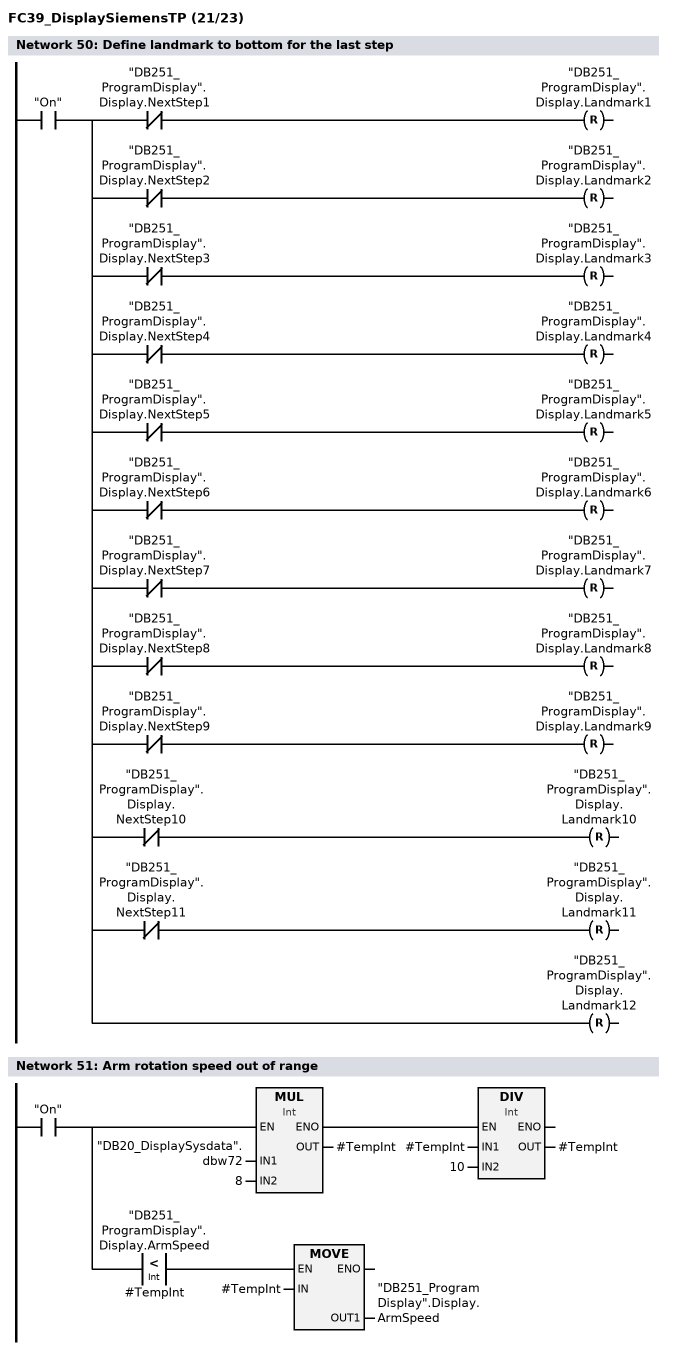
   RUNG wire#powerrail
      Contact( "On" )
      wire#w1
      I_Contact( "DB251_ProgramDisplay".Display.NextStep1 )
      R_Coil( "DB251_ProgramDisplay".Display.Landmark1 )
   END_RUNG
   RUNG wire#w1
      I_Contact( "DB251_ProgramDisplay".Display.NextStep2 )
      R_Coil( "DB251_ProgramDisplay".Display.Landmark2 )
   END_RUNG
   RUNG wire#w1
      I_Contact( "DB251_ProgramDisplay".Display.NextStep3 )
      R_Coil( "DB251_ProgramDisplay".Display.Landmark3 )
   END_RUNG
   RUNG wire#w1
      I_Contact( "DB251_ProgramDisplay".Display.NextStep4 )
      R_Coil( "DB251_ProgramDisplay".Display.Landmark4 )
   END_RUNG
   RUNG wire#w1
      I_Contact( "DB251_ProgramDisplay".Display.NextStep5 )
      R_Coil( "DB251_ProgramDisplay".Display.Landmark5 )
   END_RUNG
   RUNG wire#w1
      I_Contact( "DB251_ProgramDisplay".Display.NextStep6 )
      R_Coil( "DB251_ProgramDisplay".Display.Landmark6 )
   END_RUNG
   RUNG wire#w1
      I_Contact( "DB251_ProgramDisplay".Display.NextStep7 )
      R_Coil( "DB251_ProgramDisplay".Display.Landmark7 )
   END_RUNG
   RUNG wire#w1
      I_Contact( "DB251_ProgramDisplay".Display.NextStep8 )
      R_Coil( "DB251_ProgramDisplay".Display.Landmark8 )
   END_RUNG
   RUNG wire#w1
      I_Contact( "DB251_ProgramDisplay".Display.NextStep9 )
      R_Coil( "DB251_ProgramDisplay".Display.Landmark9 )
   END_RUNG
   RUNG wire#w1
      I_Contact( "DB251_ProgramDisplay".Display.NextStep10 )
      R_Coil( "DB251_ProgramDisplay".Display.Landmark10 )
   END_RUNG
   RUNG wire#w1
      I_Contact( "DB251_ProgramDisplay".Display.NextStep11 )
      R_Coil( "DB251_ProgramDisplay".Display.Landmark11 )
   END_RUNG
   RUNG wire#w1
      R_Coil( "DB251_ProgramDisplay".Display.Landmark12 )
   END_RUNG
   // the same network as SCL:
   IF "On" AND NOT "DB251_ProgramDisplay".Display.NextStep1 THEN
       "DB251_ProgramDisplay".Display.Landmark1 := FALSE;
   END_IF;
   IF "On" AND NOT "DB251_ProgramDisplay".Display.NextStep2 THEN
       "DB251_ProgramDisplay".Display.Landmark2 := FALSE;
   END_IF;
   IF "On" AND NOT "DB251_ProgramDisplay".Display.NextStep3 THEN
       "DB251_ProgramDisplay".Display.Landmark3 := FALSE;
   END_IF;
   IF "On" AND NOT "DB251_ProgramDisplay".Display.NextStep4 THEN
       "DB251_ProgramDisplay".Display.Landmark4 := FALSE;
   END_IF;
   IF "On" AND NOT "DB251_ProgramDisplay".Display.NextStep5 THEN
       "DB251_ProgramDisplay".Display.Landmark5 := FALSE;
   END_IF;
   IF "On" AND NOT "DB251_ProgramDisplay".Display.NextStep6 THEN
       "DB251_ProgramDisplay".Display.Landmark6 := FALSE;
   END_IF;
   IF "On" AND NOT "DB251_ProgramDisplay".Display.NextStep7 THEN
       "DB251_ProgramDisplay".Display.Landmark7 := FALSE;
   END_IF;
   IF "On" AND NOT "DB251_ProgramDisplay".Display.NextStep8 THEN
       "DB251_ProgramDisplay".Display.Landmark8 := FALSE;
   END_IF;
   IF "On" AND NOT "DB251_ProgramDisplay".Display.NextStep9 THEN
       "DB251_ProgramDisplay".Display.Landmark9 := FALSE;
   END_IF;
   IF "On" AND NOT "DB251_ProgramDisplay".Display.NextStep10 THEN
       "DB251_ProgramDisplay".Display.Landmark10 := FALSE;
   END_IF;
   IF "On" AND NOT "DB251_ProgramDisplay".Display.NextStep11 THEN
       "DB251_ProgramDisplay".Display.Landmark11 := FALSE;
   END_IF;
   IF "On" THEN "DB251_ProgramDisplay".Display.Landmark12 := FALSE; END_IF;
END_REGION

REGION Network 51: Arm rotation speed out of range
   RUNG wire#powerrail
      Contact( "On" )
      wire#w1
      { S7_Templates := "SrcType := Int"; S7_GenerateENO := "TRUE" } Mul(in1 := "DB20_DisplaySysdata".dbw72, in2 := 8, out => #TempInt)
      { S7_Templates := "SrcType := Int"; S7_GenerateENO := "TRUE" } Div(in1 := #TempInt, in2 := 10, out => #TempInt)
   END_RUNG
   RUNG wire#w1
      { S7_Templates := "SrcType := Int" } LT_Contact(in1 := "DB251_ProgramDisplay".Display.ArmSpeed, in2 := #TempInt)
      { S7_GenerateENO := "TRUE" } Move(in := #TempInt, out1 => "DB251_ProgramDisplay".Display.ArmSpeed)
   END_RUNG
   // the same network as SCL:
   // ENO of a box is taken as its EN; it also drops when the box reports an error
   IF "On" THEN
       #TempInt := "DB20_DisplaySysdata".dbw72 * 8;
       #TempInt := #TempInt / 10;
   END_IF;
   IF "On" AND ("DB251_ProgramDisplay".Display.ArmSpeed < #TempInt) THEN
       "DB251_ProgramDisplay".Display.ArmSpeed := #TempInt;
   END_IF;
END_REGION

REGION Network 52: Next step for spool carriage height 12 (0=End 1=Next)
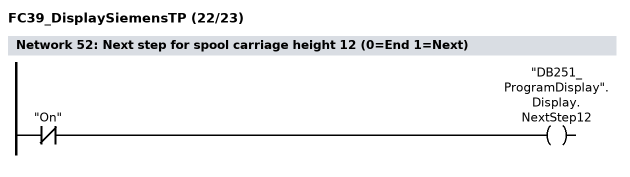
   RUNG wire#powerrail
      I_Contact( "On" )
      Coil( "DB251_ProgramDisplay".Display.NextStep12 )
   END_RUNG
   // the same network as SCL:
   "DB251_ProgramDisplay".Display.NextStep12 := NOT "On";
END_REGION

REGION Network 53
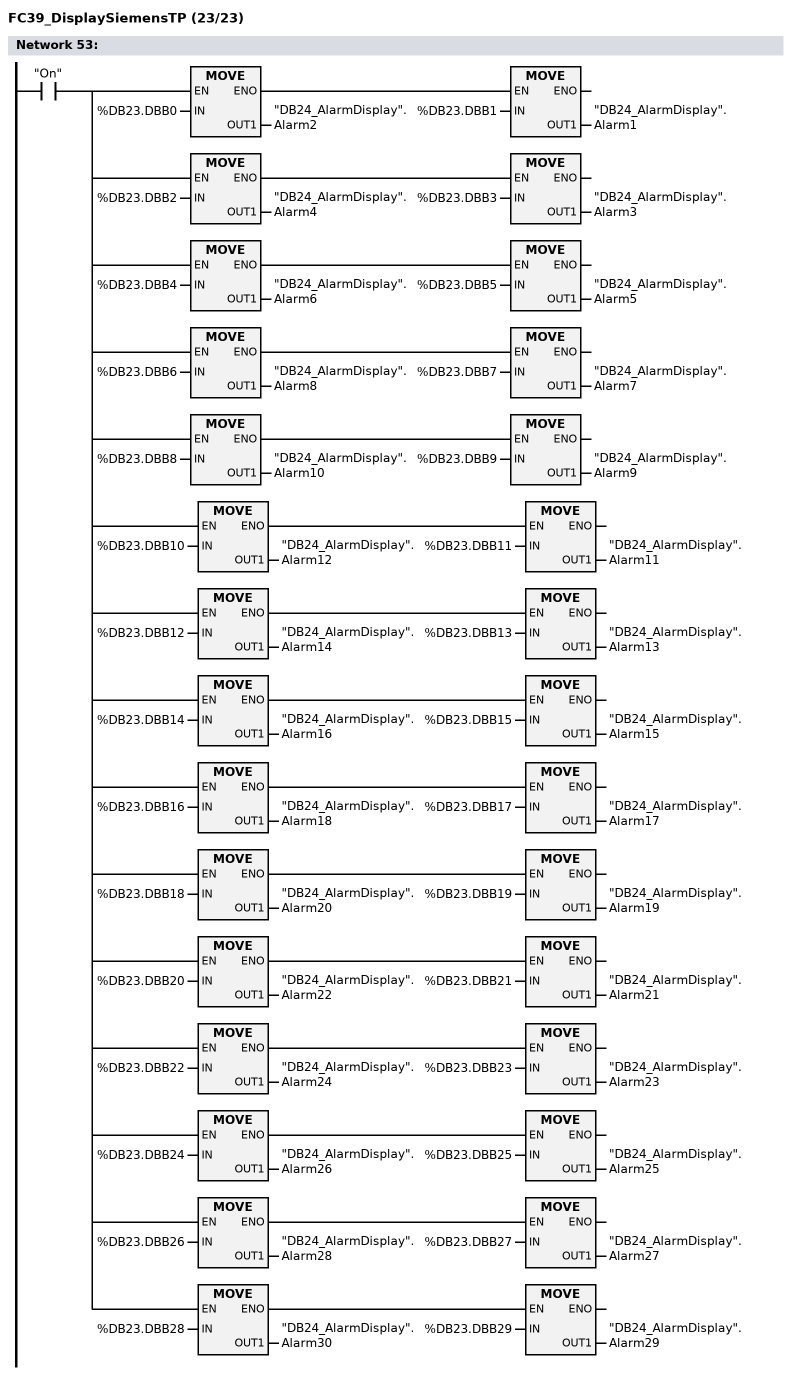
   RUNG wire#powerrail
      Contact( "On" )
      wire#w1
      { S7_GenerateENO := "TRUE" } Move(in := %DB23.DBB0, out1 => "DB24_AlarmDisplay".Alarm2)
      { S7_GenerateENO := "TRUE" } Move(in := %DB23.DBB1, out1 => "DB24_AlarmDisplay".Alarm1)
   END_RUNG
   RUNG wire#w1
      { S7_GenerateENO := "TRUE" } Move(in := %DB23.DBB2, out1 => "DB24_AlarmDisplay".Alarm4)
      { S7_GenerateENO := "TRUE" } Move(in := %DB23.DBB3, out1 => "DB24_AlarmDisplay".Alarm3)
   END_RUNG
   RUNG wire#w1
      { S7_GenerateENO := "TRUE" } Move(in := %DB23.DBB4, out1 => "DB24_AlarmDisplay".Alarm6)
      { S7_GenerateENO := "TRUE" } Move(in := %DB23.DBB5, out1 => "DB24_AlarmDisplay".Alarm5)
   END_RUNG
   RUNG wire#w1
      { S7_GenerateENO := "TRUE" } Move(in := %DB23.DBB6, out1 => "DB24_AlarmDisplay".Alarm8)
      { S7_GenerateENO := "TRUE" } Move(in := %DB23.DBB7, out1 => "DB24_AlarmDisplay".Alarm7)
   END_RUNG
   RUNG wire#w1
      { S7_GenerateENO := "TRUE" } Move(in := %DB23.DBB8, out1 => "DB24_AlarmDisplay".Alarm10)
      { S7_GenerateENO := "TRUE" } Move(in := %DB23.DBB9, out1 => "DB24_AlarmDisplay".Alarm9)
   END_RUNG
   RUNG wire#w1
      { S7_GenerateENO := "TRUE" } Move(in := %DB23.DBB10, out1 => "DB24_AlarmDisplay".Alarm12)
      { S7_GenerateENO := "TRUE" } Move(in := %DB23.DBB11, out1 => "DB24_AlarmDisplay".Alarm11)
   END_RUNG
   RUNG wire#w1
      { S7_GenerateENO := "TRUE" } Move(in := %DB23.DBB12, out1 => "DB24_AlarmDisplay".Alarm14)
      { S7_GenerateENO := "TRUE" } Move(in := %DB23.DBB13, out1 => "DB24_AlarmDisplay".Alarm13)
   END_RUNG
   RUNG wire#w1
      { S7_GenerateENO := "TRUE" } Move(in := %DB23.DBB14, out1 => "DB24_AlarmDisplay".Alarm16)
      { S7_GenerateENO := "TRUE" } Move(in := %DB23.DBB15, out1 => "DB24_AlarmDisplay".Alarm15)
   END_RUNG
   RUNG wire#w1
      { S7_GenerateENO := "TRUE" } Move(in := %DB23.DBB16, out1 => "DB24_AlarmDisplay".Alarm18)
      { S7_GenerateENO := "TRUE" } Move(in := %DB23.DBB17, out1 => "DB24_AlarmDisplay".Alarm17)
   END_RUNG
   RUNG wire#w1
      { S7_GenerateENO := "TRUE" } Move(in := %DB23.DBB18, out1 => "DB24_AlarmDisplay".Alarm20)
      { S7_GenerateENO := "TRUE" } Move(in := %DB23.DBB19, out1 => "DB24_AlarmDisplay".Alarm19)
   END_RUNG
   RUNG wire#w1
      { S7_GenerateENO := "TRUE" } Move(in := %DB23.DBB20, out1 => "DB24_AlarmDisplay".Alarm22)
      { S7_GenerateENO := "TRUE" } Move(in := %DB23.DBB21, out1 => "DB24_AlarmDisplay".Alarm21)
   END_RUNG
   RUNG wire#w1
      { S7_GenerateENO := "TRUE" } Move(in := %DB23.DBB22, out1 => "DB24_AlarmDisplay".Alarm24)
      { S7_GenerateENO := "TRUE" } Move(in := %DB23.DBB23, out1 => "DB24_AlarmDisplay".Alarm23)
   END_RUNG
   RUNG wire#w1
      { S7_GenerateENO := "TRUE" } Move(in := %DB23.DBB24, out1 => "DB24_AlarmDisplay".Alarm26)
      { S7_GenerateENO := "TRUE" } Move(in := %DB23.DBB25, out1 => "DB24_AlarmDisplay".Alarm25)
   END_RUNG
   RUNG wire#w1
      { S7_GenerateENO := "TRUE" } Move(in := %DB23.DBB26, out1 => "DB24_AlarmDisplay".Alarm28)
      { S7_GenerateENO := "TRUE" } Move(in := %DB23.DBB27, out1 => "DB24_AlarmDisplay".Alarm27)
   END_RUNG
   RUNG wire#w1
      { S7_GenerateENO := "TRUE" } Move(in := %DB23.DBB28, out1 => "DB24_AlarmDisplay".Alarm30)
      { S7_GenerateENO := "TRUE" } Move(in := %DB23.DBB29, out1 => "DB24_AlarmDisplay".Alarm29)
   END_RUNG
   // the same network as SCL:
   // ENO of a box is taken as its EN; it also drops when the box reports an error
   IF "On" THEN
       "DB24_AlarmDisplay".Alarm2 := %DB23.DBB0;
       "DB24_AlarmDisplay".Alarm1 := %DB23.DBB1;
       "DB24_AlarmDisplay".Alarm4 := %DB23.DBB2;
       "DB24_AlarmDisplay".Alarm3 := %DB23.DBB3;
       "DB24_AlarmDisplay".Alarm6 := %DB23.DBB4;
       "DB24_AlarmDisplay".Alarm5 := %DB23.DBB5;
       "DB24_AlarmDisplay".Alarm8 := %DB23.DBB6;
       "DB24_AlarmDisplay".Alarm7 := %DB23.DBB7;
       "DB24_AlarmDisplay".Alarm10 := %DB23.DBB8;
       "DB24_AlarmDisplay".Alarm9 := %DB23.DBB9;
       "DB24_AlarmDisplay".Alarm12 := %DB23.DBB10;
       "DB24_AlarmDisplay".Alarm11 := %DB23.DBB11;
       "DB24_AlarmDisplay".Alarm14 := %DB23.DBB12;
       "DB24_AlarmDisplay".Alarm13 := %DB23.DBB13;
       "DB24_AlarmDisplay".Alarm16 := %DB23.DBB14;
       "DB24_AlarmDisplay".Alarm15 := %DB23.DBB15;
       "DB24_AlarmDisplay".Alarm18 := %DB23.DBB16;
       "DB24_AlarmDisplay".Alarm17 := %DB23.DBB17;
       "DB24_AlarmDisplay".Alarm20 := %DB23.DBB18;
       "DB24_AlarmDisplay".Alarm19 := %DB23.DBB19;
       "DB24_AlarmDisplay".Alarm22 := %DB23.DBB20;
       "DB24_AlarmDisplay".Alarm21 := %DB23.DBB21;
       "DB24_AlarmDisplay".Alarm24 := %DB23.DBB22;
       "DB24_AlarmDisplay".Alarm23 := %DB23.DBB23;
       "DB24_AlarmDisplay".Alarm26 := %DB23.DBB24;
       "DB24_AlarmDisplay".Alarm25 := %DB23.DBB25;
       "DB24_AlarmDisplay".Alarm28 := %DB23.DBB26;
       "DB24_AlarmDisplay".Alarm27 := %DB23.DBB27;
       "DB24_AlarmDisplay".Alarm30 := %DB23.DBB28;
       "DB24_AlarmDisplay".Alarm29 := %DB23.DBB29;
   END_IF;
END_REGION
END_FUNCTION

FUNCTION "FC105_GreyBarReset" : Void   // FC105, LAD
TITLE = Reset grey bar program data
{ S7_Optimized_Access := 'TRUE' }
VERSION : 0.1
// stored: AutoNumber false, IsIECCheckEnabled false, SetENOAutomatically false, UDAEnableTagReadback false
BEGIN

REGION Network 1: Reset grey bar program data
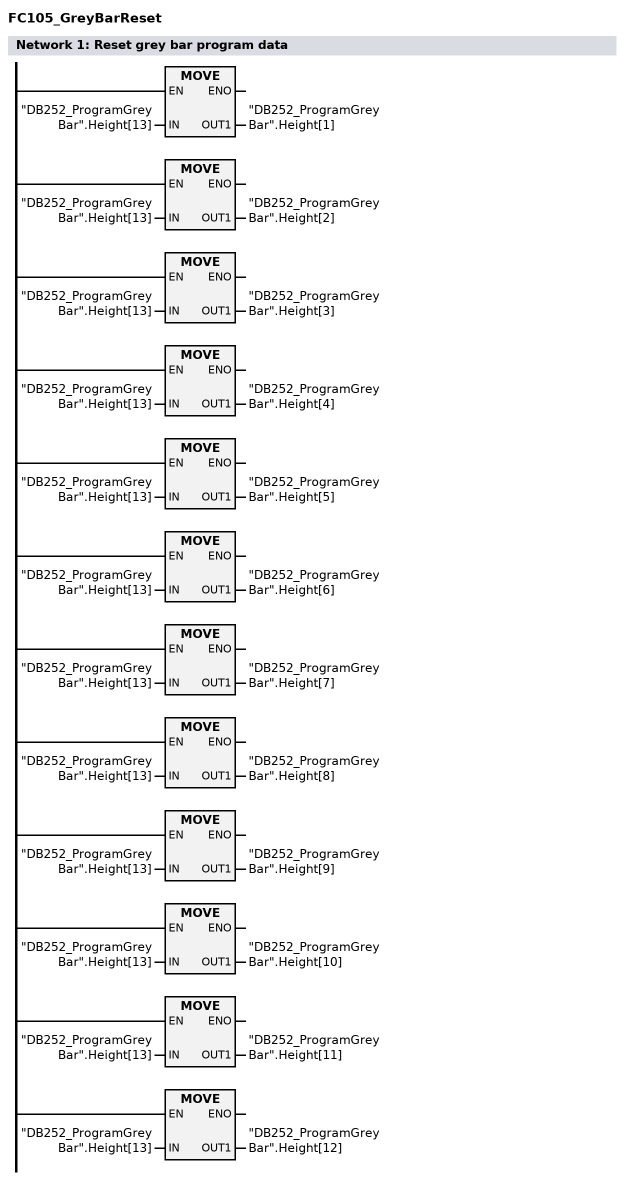
   RUNG wire#powerrail
      { S7_GenerateENO := "TRUE" } Move(in := "DB252_ProgramGreyBar".Height[13], out1 => "DB252_ProgramGreyBar".Height[1])
   END_RUNG
   RUNG wire#powerrail
      { S7_GenerateENO := "TRUE" } Move(in := "DB252_ProgramGreyBar".Height[13], out1 => "DB252_ProgramGreyBar".Height[2])
   END_RUNG
   RUNG wire#powerrail
      { S7_GenerateENO := "TRUE" } Move(in := "DB252_ProgramGreyBar".Height[13], out1 => "DB252_ProgramGreyBar".Height[3])
   END_RUNG
   RUNG wire#powerrail
      { S7_GenerateENO := "TRUE" } Move(in := "DB252_ProgramGreyBar".Height[13], out1 => "DB252_ProgramGreyBar".Height[4])
   END_RUNG
   RUNG wire#powerrail
      { S7_GenerateENO := "TRUE" } Move(in := "DB252_ProgramGreyBar".Height[13], out1 => "DB252_ProgramGreyBar".Height[5])
   END_RUNG
   RUNG wire#powerrail
      { S7_GenerateENO := "TRUE" } Move(in := "DB252_ProgramGreyBar".Height[13], out1 => "DB252_ProgramGreyBar".Height[6])
   END_RUNG
   RUNG wire#powerrail
      { S7_GenerateENO := "TRUE" } Move(in := "DB252_ProgramGreyBar".Height[13], out1 => "DB252_ProgramGreyBar".Height[7])
   END_RUNG
   RUNG wire#powerrail
      { S7_GenerateENO := "TRUE" } Move(in := "DB252_ProgramGreyBar".Height[13], out1 => "DB252_ProgramGreyBar".Height[8])
   END_RUNG
   RUNG wire#powerrail
      { S7_GenerateENO := "TRUE" } Move(in := "DB252_ProgramGreyBar".Height[13], out1 => "DB252_ProgramGreyBar".Height[9])
   END_RUNG
   RUNG wire#powerrail
      { S7_GenerateENO := "TRUE" } Move(in := "DB252_ProgramGreyBar".Height[13], out1 => "DB252_ProgramGreyBar".Height[10])
   END_RUNG
   RUNG wire#powerrail
      { S7_GenerateENO := "TRUE" } Move(in := "DB252_ProgramGreyBar".Height[13], out1 => "DB252_ProgramGreyBar".Height[11])
   END_RUNG
   RUNG wire#powerrail
      { S7_GenerateENO := "TRUE" } Move(in := "DB252_ProgramGreyBar".Height[13], out1 => "DB252_ProgramGreyBar".Height[12])
   END_RUNG
   // the same network as SCL:
   "DB252_ProgramGreyBar".Height[1] := "DB252_ProgramGreyBar".Height[13];
   "DB252_ProgramGreyBar".Height[2] := "DB252_ProgramGreyBar".Height[13];
   "DB252_ProgramGreyBar".Height[3] := "DB252_ProgramGreyBar".Height[13];
   "DB252_ProgramGreyBar".Height[4] := "DB252_ProgramGreyBar".Height[13];
   "DB252_ProgramGreyBar".Height[5] := "DB252_ProgramGreyBar".Height[13];
   "DB252_ProgramGreyBar".Height[6] := "DB252_ProgramGreyBar".Height[13];
   "DB252_ProgramGreyBar".Height[7] := "DB252_ProgramGreyBar".Height[13];
   "DB252_ProgramGreyBar".Height[8] := "DB252_ProgramGreyBar".Height[13];
   "DB252_ProgramGreyBar".Height[9] := "DB252_ProgramGreyBar".Height[13];
   "DB252_ProgramGreyBar".Height[10] := "DB252_ProgramGreyBar".Height[13];
   "DB252_ProgramGreyBar".Height[11] := "DB252_ProgramGreyBar".Height[13];
   "DB252_ProgramGreyBar".Height[12] := "DB252_ProgramGreyBar".Height[13];
END_REGION
END_FUNCTION

FUNCTION "FC41_NoRopeUnit" : Void   // FC41, LAD
TITLE = No rope unit
{ S7_Optimized_Access := 'FALSE' }
AUTHOR : Robopac
VERSION : 0.0
// stored: AutoNumber false, IsIECCheckEnabled false, SetENOAutomatically false, UDAEnableTagReadback false
BEGIN

REGION Network 1: RopeUnitOk1: Rope unit open
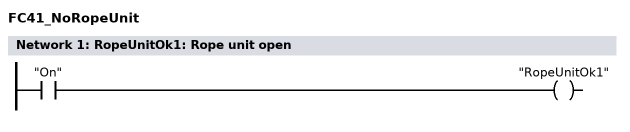
   RUNG wire#powerrail
      Contact( "On" )
      Coil( "RopeUnitOk1" )
   END_RUNG
   // the same network as SCL:
   "RopeUnitOk1" := "On";
END_REGION
END_FUNCTION

FUNCTION "FC05_TechnoplatOutput" : Void   // FC5, LAD
TITLE = Machine output
{ S7_Optimized_Access := 'FALSE' }
AUTHOR : Robopac
VERSION : 0.0
// stored: AutoNumber false, IsIECCheckEnabled false, SetENOAutomatically false, UDAEnableTagReadback false
   VAR_INPUT
      PHASE : Bool;
      FASTSPEED : Bool;
   END_VAR
   VAR_TEMP
      SuppSpeed : Bool;
      wTemp : Int;
      DwTemp : DInt;
      wTemp2 : Int;
      wTemp3 : Int;
      U201_START : Bool;
      U201_DIR : Bool;
      U201_SP : Int;
      U221_START : Bool;
      U221_DIR : Bool;
      U221_SP : Int;
      DwTemp2 : DInt;
   END_VAR
   VAR_TEMP   // added for the SCL form of the ladder/FBD networks
      _w1 : Bool;
   END_VAR
BEGIN

REGION Network 1: Emergency mode lamp (Helix)
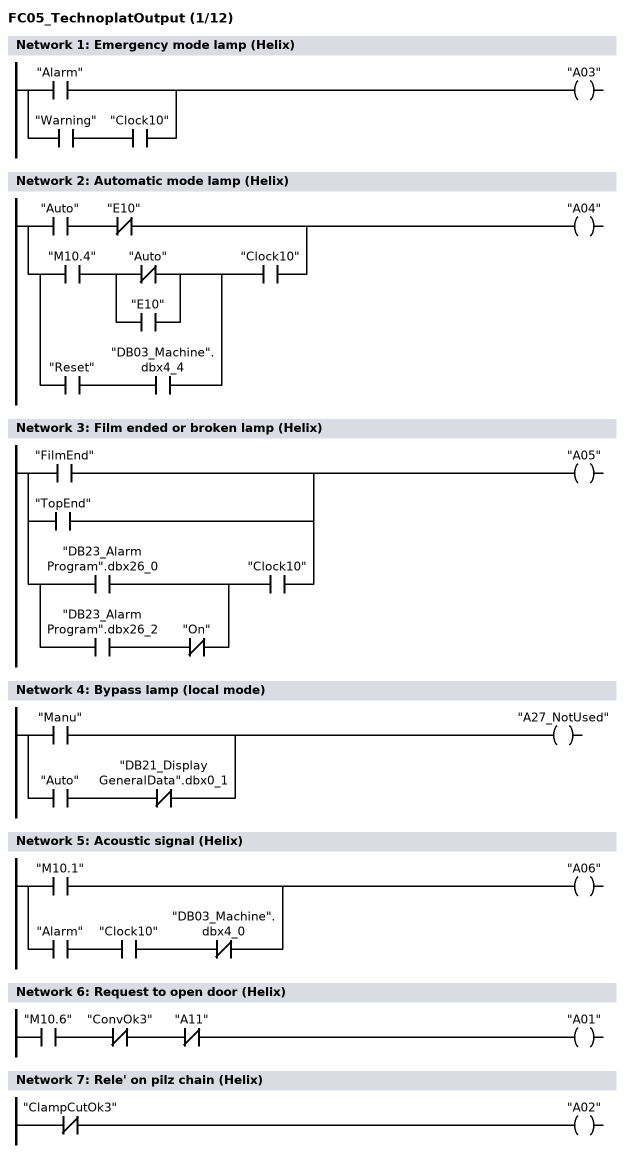
   RUNG wire#powerrail
      Contact( "Alarm" )
      wire#w1
      Coil( "A03" )
   END_RUNG
   RUNG wire#powerrail
      Contact( "Warning" )
      Contact( "Clock10" )
   END_RUNG wire#w1
   // the same network as SCL:
   "A03" := "Alarm" OR ("Warning" AND "Clock10");
END_REGION

REGION Network 2: Automatic mode lamp (Helix)
   RUNG wire#powerrail
      Contact( "Auto" )
      I_Contact( "E10" )
      wire#w1
      Coil( "A04" )
   END_RUNG
   RUNG wire#powerrail
      Contact( "M10.4" )
      wire#w2
      I_Contact( "Auto" )
      wire#w3
      Contact( "Clock10" )
   END_RUNG wire#w1
   RUNG wire#w2
      Contact( "E10" )
   END_RUNG wire#w3
   RUNG wire#powerrail
      Contact( "Reset" )
      Contact( "DB03_Machine".dbx4_4 )
   END_RUNG wire#w3
   // the same network as SCL:
   "A04" := ("Auto" AND NOT "E10") OR ((("M10.4" AND (NOT "Auto" OR "E10")) OR ("Reset" AND "DB03_Machine".dbx4_4)) AND "Clock10");
END_REGION

REGION Network 3: Film ended or broken lamp (Helix)
   RUNG wire#powerrail
      Contact( "FilmEnd" )
      wire#w1
      Coil( "A05" )
   END_RUNG
   RUNG wire#powerrail
      Contact( "TopEnd" )
   END_RUNG wire#w1
   RUNG wire#powerrail
      Contact( "DB23_AlarmProgram".dbx26_0 )
      wire#w2
      Contact( "Clock10" )
   END_RUNG wire#w1
   RUNG wire#powerrail
      Contact( "DB23_AlarmProgram".dbx26_2 )
      I_Contact( "On" )
   END_RUNG wire#w2
   // the same network as SCL:
   "A05" := "FilmEnd" OR "TopEnd" OR (("DB23_AlarmProgram".dbx26_0 OR ("DB23_AlarmProgram".dbx26_2 AND NOT "On")) AND "Clock10");
END_REGION

REGION Network 4: Bypass lamp (local mode)
   RUNG wire#powerrail
      Contact( "Manu" )
      wire#w1
      Coil( "A27_NotUsed" )
   END_RUNG
   RUNG wire#powerrail
      Contact( "Auto" )
      I_Contact( "DB21_DisplayGeneralData".dbx0_1 )
   END_RUNG wire#w1
   // the same network as SCL:
   "A27_NotUsed" := "Manu" OR ("Auto" AND NOT "DB21_DisplayGeneralData".dbx0_1);
END_REGION

REGION Network 5: Acoustic signal (Helix)
   RUNG wire#powerrail
      Contact( "M10.1" )
      wire#w1
      Coil( "A06" )
   END_RUNG
   RUNG wire#powerrail
      Contact( "Alarm" )
      Contact( "Clock10" )
      I_Contact( "DB03_Machine".dbx4_0 )
   END_RUNG wire#w1
   // the same network as SCL:
   "A06" := "M10.1" OR ("Alarm" AND "Clock10" AND NOT "DB03_Machine".dbx4_0);
END_REGION

REGION Network 6: Request to open door (Helix)
   RUNG wire#powerrail
      Contact( "M10.6" )
      I_Contact( "ConvOk3" )
      I_Contact( "A11" )
      Coil( "A01" )
   END_RUNG
   // the same network as SCL:
   "A01" := "M10.6" AND NOT "ConvOk3" AND NOT "A11";
END_REGION

REGION Network 7: Rele' on pilz chain (Helix)
   RUNG wire#powerrail
      I_Contact( "ClampCutOk3" )
      Coil( "A02" )
   END_RUNG
   // the same network as SCL:
   "A02" := NOT "ClampCutOk3";
END_REGION

REGION Network 8: Table rotation forward
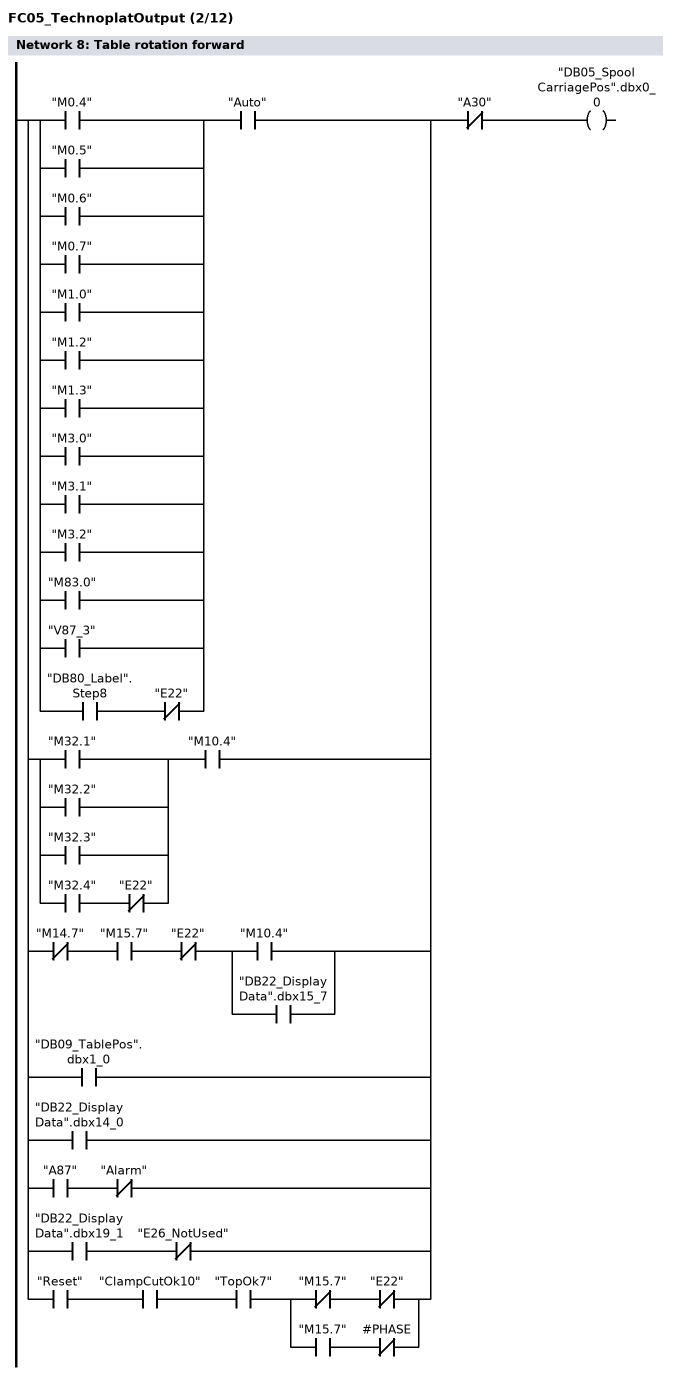
   RUNG wire#powerrail
      Contact( "M0.4" )
      wire#w1
      Contact( "Auto" )
      wire#w2
      I_Contact( "A30" )
      Coil( "DB05_SpoolCarriagePos".dbx0_0 )
   END_RUNG
   RUNG wire#powerrail
      Contact( "M0.5" )
   END_RUNG wire#w1
   RUNG wire#powerrail
      Contact( "M0.6" )
   END_RUNG wire#w1
   RUNG wire#powerrail
      Contact( "M0.7" )
   END_RUNG wire#w1
   RUNG wire#powerrail
      Contact( "M1.0" )
   END_RUNG wire#w1
   RUNG wire#powerrail
      Contact( "M1.2" )
   END_RUNG wire#w1
   RUNG wire#powerrail
      Contact( "M1.3" )
   END_RUNG wire#w1
   RUNG wire#powerrail
      Contact( "M3.0" )
   END_RUNG wire#w1
   RUNG wire#powerrail
      Contact( "M3.1" )
   END_RUNG wire#w1
   RUNG wire#powerrail
      Contact( "M3.2" )
   END_RUNG wire#w1
   RUNG wire#powerrail
      Contact( "M83.0" )
   END_RUNG wire#w1
   RUNG wire#powerrail
      Contact( "V87_3" )
   END_RUNG wire#w1
   RUNG wire#powerrail
      Contact( "DB80_Label".Step8 )
      I_Contact( "E22" )
   END_RUNG wire#w1
   RUNG wire#powerrail
      Contact( "M32.1" )
      wire#w3
      Contact( "M10.4" )
   END_RUNG wire#w2
   RUNG wire#powerrail
      Contact( "M32.2" )
   END_RUNG wire#w3
   RUNG wire#powerrail
      Contact( "M32.3" )
   END_RUNG wire#w3
   RUNG wire#powerrail
      Contact( "M32.4" )
      I_Contact( "E22" )
   END_RUNG wire#w3
   RUNG wire#powerrail
      I_Contact( "M14.7" )
      Contact( "M15.7" )
      I_Contact( "E22" )
      wire#w4
      Contact( "M10.4" )
   END_RUNG wire#w2
   RUNG wire#w4
      Contact( "DB22_DisplayData".dbx15_7 )
   END_RUNG wire#w2
   RUNG wire#powerrail
      Contact( "DB09_TablePos".dbx1_0 )
   END_RUNG wire#w2
   RUNG wire#powerrail
      Contact( "DB22_DisplayData".dbx14_0 )
   END_RUNG wire#w2
   RUNG wire#powerrail
      Contact( "A87" )
      I_Contact( "Alarm" )
   END_RUNG wire#w2
   RUNG wire#powerrail
      Contact( "DB22_DisplayData".dbx19_1 )
      I_Contact( "E26_NotUsed" )
   END_RUNG wire#w2
   RUNG wire#powerrail
      Contact( "Reset" )
      Contact( "ClampCutOk10" )
      Contact( "TopOk7" )
      wire#w5
      I_Contact( "M15.7" )
      I_Contact( "E22" )
   END_RUNG wire#w2
   RUNG wire#w5
      Contact( "M15.7" )
      I_Contact( #PHASE )
   END_RUNG wire#w2
   // the same network as SCL:
   "DB05_SpoolCarriagePos".dbx0_0 := ((("M0.4" OR "M0.5" OR "M0.6" OR "M0.7" OR "M1.0" OR "M1.2" OR "M1.3" OR "M3.0" OR "M3.1" OR "M3.2" OR "M83.0" OR "V87_3" OR ("DB80_Label".Step8 AND NOT "E22")) AND "Auto") OR (("M32.1" OR "M32.2" OR "M32.3" OR ("M32.4" AND NOT "E22")) AND "M10.4") OR (NOT "M14.7" AND "M15.7" AND NOT "E22" AND ("M10.4" OR "DB22_DisplayData".dbx15_7)) OR "DB09_TablePos".dbx1_0 OR "DB22_DisplayData".dbx14_0 OR ("A87" AND NOT "Alarm") OR ("DB22_DisplayData".dbx19_1 AND NOT "E26_NotUsed") OR ("Reset" AND "ClampCutOk10" AND "TopOk7" AND ((NOT "M15.7" AND NOT "E22") OR ("M15.7" AND NOT #PHASE)))) AND NOT "A30";
END_REGION

REGION Network 9: Table rotation backward
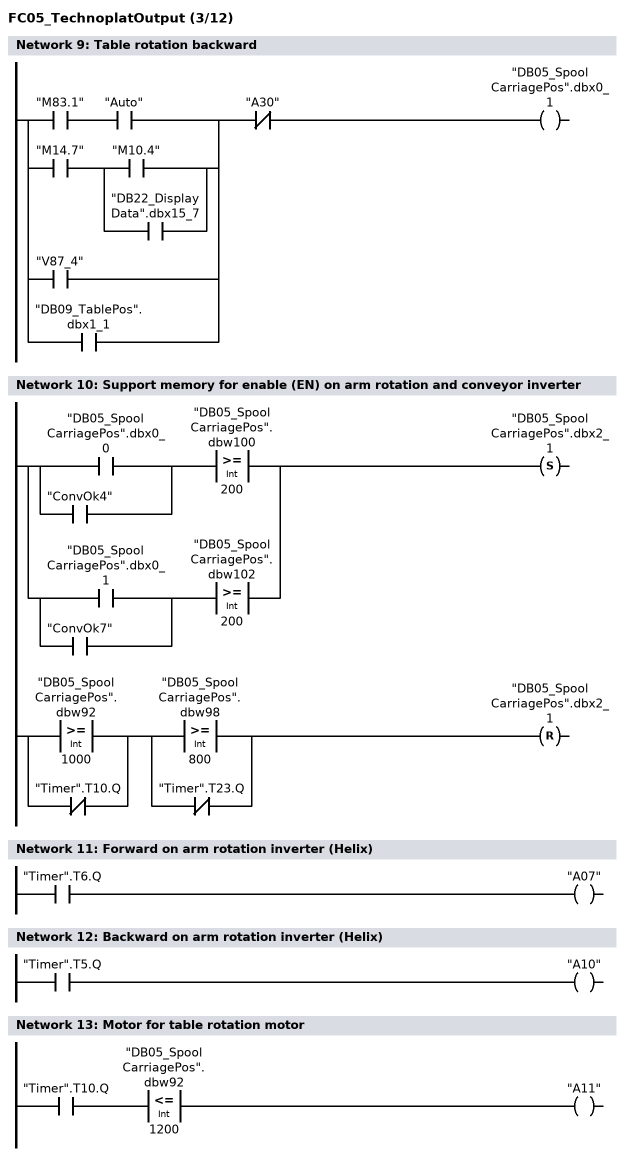
   RUNG wire#powerrail
      Contact( "M83.1" )
      Contact( "Auto" )
      wire#w1
      I_Contact( "A30" )
      Coil( "DB05_SpoolCarriagePos".dbx0_1 )
   END_RUNG
   RUNG wire#powerrail
      Contact( "M14.7" )
      wire#w2
      Contact( "M10.4" )
   END_RUNG wire#w1
   RUNG wire#w2
      Contact( "DB22_DisplayData".dbx15_7 )
   END_RUNG wire#w1
   RUNG wire#powerrail
      Contact( "V87_4" )
   END_RUNG wire#w1
   RUNG wire#powerrail
      Contact( "DB09_TablePos".dbx1_1 )
   END_RUNG wire#w1
   // the same network as SCL:
   "DB05_SpoolCarriagePos".dbx0_1 := (("M83.1" AND "Auto") OR ("M14.7" AND ("M10.4" OR "DB22_DisplayData".dbx15_7)) OR "V87_4" OR "DB09_TablePos".dbx1_1) AND NOT "A30";
END_REGION

REGION Network 10: Support memory for enable (EN) on arm rotation and conveyor inverter
   RUNG wire#powerrail
      Contact( "DB05_SpoolCarriagePos".dbx0_0 )
      wire#w1
      { S7_Templates := "SrcType := Int" } GE_Contact(in1 := "DB05_SpoolCarriagePos".dbw100, in2 := 200)
      wire#w2
      S_Coil( "DB05_SpoolCarriagePos".dbx2_1 )
   END_RUNG
   RUNG wire#powerrail
      Contact( "ConvOk4" )
   END_RUNG wire#w1
   RUNG wire#powerrail
      Contact( "DB05_SpoolCarriagePos".dbx0_1 )
      wire#w3
      { S7_Templates := "SrcType := Int" } GE_Contact(in1 := "DB05_SpoolCarriagePos".dbw102, in2 := 200)
   END_RUNG wire#w2
   RUNG wire#powerrail
      Contact( "ConvOk7" )
   END_RUNG wire#w3
   RUNG wire#powerrail
      { S7_Templates := "SrcType := Int" } GE_Contact(in1 := "DB05_SpoolCarriagePos".dbw92, in2 := 1000)
      wire#w4
      { S7_Templates := "SrcType := Int" } GE_Contact(in1 := "DB05_SpoolCarriagePos".dbw98, in2 := 800)
      wire#w5
      R_Coil( "DB05_SpoolCarriagePos".dbx2_1 )
   END_RUNG
   RUNG wire#powerrail
      I_Contact( "Timer".T10.Q )
   END_RUNG wire#w4
   RUNG wire#w4
      I_Contact( "Timer".T23.Q )
   END_RUNG wire#w5
   // the same network as SCL:
   IF (("DB05_SpoolCarriagePos".dbx0_0 OR "ConvOk4") AND ("DB05_SpoolCarriagePos".dbw100 >= 200)) OR (("DB05_SpoolCarriagePos".dbx0_1 OR "ConvOk7") AND ("DB05_SpoolCarriagePos".dbw102 >= 200)) THEN
       "DB05_SpoolCarriagePos".dbx2_1 := TRUE;
   END_IF;
   IF (("DB05_SpoolCarriagePos".dbw92 >= 1000) OR NOT "Timer".T10.Q) AND (("DB05_SpoolCarriagePos".dbw98 >= 800) OR NOT "Timer".T23.Q) THEN
       "DB05_SpoolCarriagePos".dbx2_1 := FALSE;
   END_IF;
END_REGION

REGION Network 11: Forward on arm rotation inverter (Helix)
   RUNG wire#powerrail
      Contact( "Timer".T6.Q )
      Coil( "A07" )
   END_RUNG
   // the same network as SCL:
   "A07" := "Timer".T6.Q;
END_REGION

REGION Network 12: Backward on arm rotation inverter (Helix)
   RUNG wire#powerrail
      Contact( "Timer".T5.Q )
      Coil( "A10" )
   END_RUNG
   // the same network as SCL:
   "A10" := "Timer".T5.Q;
END_REGION

REGION Network 13: Motor for table rotation motor
   RUNG wire#powerrail
      Contact( "Timer".T10.Q )
      { S7_Templates := "SrcType := Int" } LE_Contact(in1 := "DB05_SpoolCarriagePos".dbw92, in2 := 1200)
      Coil( "A11" )
   END_RUNG
   // the same network as SCL:
   "A11" := "Timer".T10.Q AND ("DB05_SpoolCarriagePos".dbw92 <= 1200);
END_REGION

REGION Network 14: Brake for table rotation motor (Technoplat)
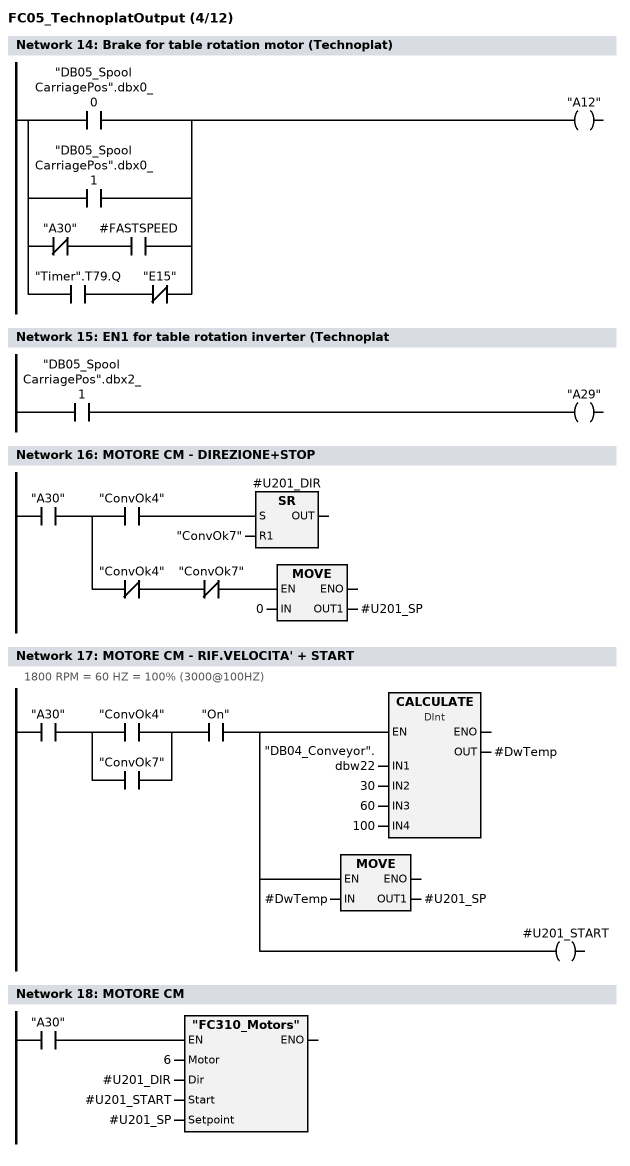
   RUNG wire#powerrail
      Contact( "DB05_SpoolCarriagePos".dbx0_0 )
      wire#w1
      Coil( "A12" )
   END_RUNG
   RUNG wire#powerrail
      Contact( "DB05_SpoolCarriagePos".dbx0_1 )
   END_RUNG wire#w1
   RUNG wire#powerrail
      I_Contact( "A30" )
      Contact( #FASTSPEED )
   END_RUNG wire#w1
   RUNG wire#powerrail
      Contact( "Timer".T79.Q )
      I_Contact( "E15" )
   END_RUNG wire#w1
   // the same network as SCL:
   "A12" := "DB05_SpoolCarriagePos".dbx0_0 OR "DB05_SpoolCarriagePos".dbx0_1 OR (NOT "A30" AND #FASTSPEED) OR ("Timer".T79.Q AND NOT "E15");
END_REGION

REGION Network 15: EN1 for table rotation inverter (Technoplat
   RUNG wire#powerrail
      Contact( "DB05_SpoolCarriagePos".dbx2_1 )
      Coil( "A29" )
   END_RUNG
   // the same network as SCL:
   "A29" := "DB05_SpoolCarriagePos".dbx2_1;
END_REGION

REGION Network 16: MOTORE CM - DIREZIONE+STOP
   RUNG wire#powerrail
      Contact( "A30" )
      wire#w1
      Contact( "ConvOk4" )
      S_SR(operand := #U201_DIR, r1 := "ConvOk7")
   END_RUNG
   RUNG wire#w1
      I_Contact( "ConvOk4" )
      I_Contact( "ConvOk7" )
      Move(in := 0, out1 => #U201_SP)
   END_RUNG
   // the same network as SCL:
   IF "A30" AND "ConvOk4" THEN
       #U201_DIR := TRUE;   // SR flip-flop
   END_IF;
   IF "ConvOk7" THEN #U201_DIR := FALSE; END_IF;
   IF "A30" AND NOT "ConvOk4" AND NOT "ConvOk7" THEN #U201_SP := 0; END_IF;
END_REGION

REGION Network 17: MOTORE CM - RIF.VELOCITA' + START
   // 1800 RPM = 60 HZ = 100% (3000@100HZ)
   RUNG wire#powerrail
      Contact( "A30" )
      wire#w1
      Contact( "ConvOk4" )
      wire#w2
      Contact( "On" )
      wire#w3
      { S7_Templates := "SrcType := DInt"; S7_Expression := "(IN1*IN2*IN3)/IN4" } Calculate(in1 := "DB04_Conveyor".dbw22, in2 := 30, in3 := 60, in4 := 100, out => #DwTemp)
   END_RUNG
   RUNG wire#w1
      Contact( "ConvOk7" )
   END_RUNG wire#w2
   RUNG wire#w3
      Move(in := #DwTemp, out1 => #U201_SP)
   END_RUNG
   RUNG wire#w3
      Coil( #U201_START )
   END_RUNG
   // the same network as SCL:
   #_w1 := "A30" AND ("ConvOk4" OR "ConvOk7") AND "On";
   IF #_w1 THEN
       #DwTemp := ("DB04_Conveyor".dbw22*30*60)/100;
       #U201_SP := #DwTemp;
   END_IF;
   #U201_START := #_w1;
END_REGION

REGION Network 18: MOTORE CM
   RUNG wire#powerrail
      Contact( "A30" )
      "FC310_Motors"(Motor := 6, Dir := #U201_DIR, Start := #U201_START, Setpoint := #U201_SP)
   END_RUNG
   // the same network as SCL:
   IF "A30" THEN
       "FC310_Motors"(Motor := 6, Dir := #U201_DIR, Start := #U201_START, Setpoint := #U201_SP);
   END_IF;
END_REGION

REGION Network 19: Positioning command for OFF3 U201 (ON=normal functioning/OFF fast stop)
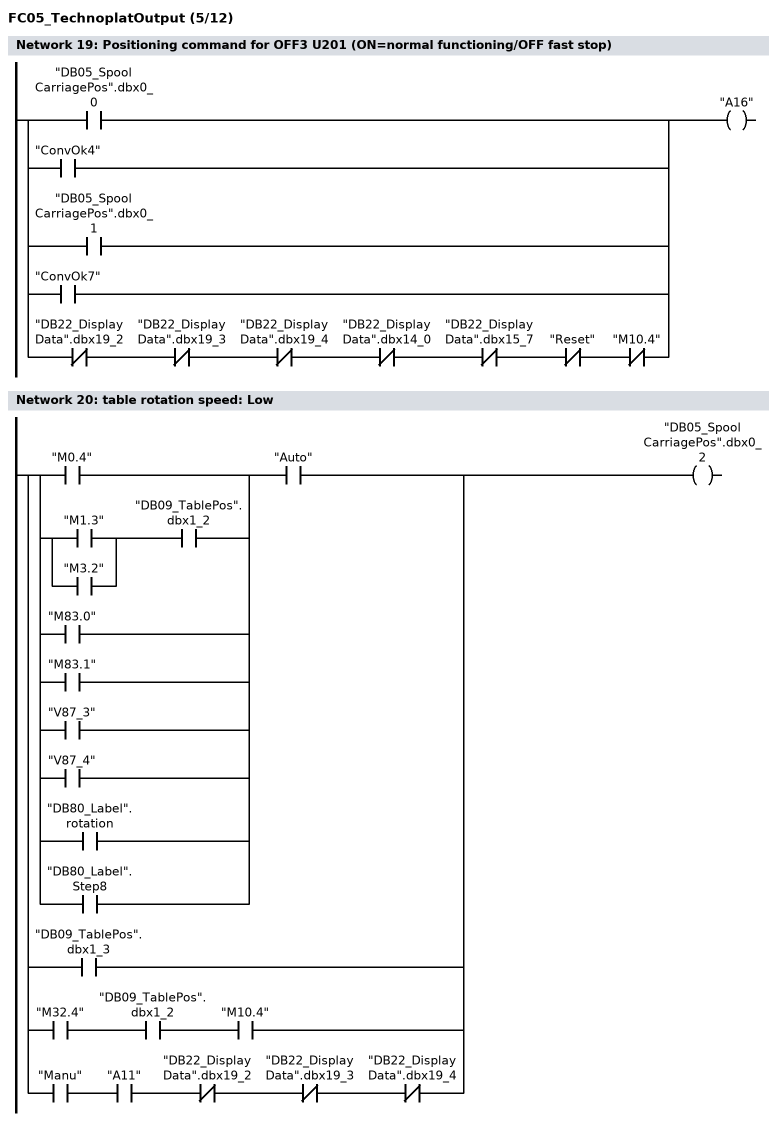
   RUNG wire#powerrail
      Contact( "DB05_SpoolCarriagePos".dbx0_0 )
      wire#w1
      Coil( "A16" )
   END_RUNG
   RUNG wire#powerrail
      Contact( "ConvOk4" )
   END_RUNG wire#w1
   RUNG wire#powerrail
      Contact( "DB05_SpoolCarriagePos".dbx0_1 )
   END_RUNG wire#w1
   RUNG wire#powerrail
      Contact( "ConvOk7" )
   END_RUNG wire#w1
   RUNG wire#powerrail
      I_Contact( "DB22_DisplayData".dbx19_2 )
      I_Contact( "DB22_DisplayData".dbx19_3 )
      I_Contact( "DB22_DisplayData".dbx19_4 )
      I_Contact( "DB22_DisplayData".dbx14_0 )
      I_Contact( "DB22_DisplayData".dbx15_7 )
      I_Contact( "Reset" )
      I_Contact( "M10.4" )
   END_RUNG wire#w1
   // the same network as SCL:
   "A16" := "DB05_SpoolCarriagePos".dbx0_0 OR "ConvOk4" OR "DB05_SpoolCarriagePos".dbx0_1 OR "ConvOk7" OR (NOT "DB22_DisplayData".dbx19_2 AND NOT "DB22_DisplayData".dbx19_3 AND NOT "DB22_DisplayData".dbx19_4 AND NOT "DB22_DisplayData".dbx14_0 AND NOT "DB22_DisplayData".dbx15_7 AND NOT "Reset" AND NOT "M10.4");
END_REGION

REGION Network 20: table rotation speed: Low
   RUNG wire#powerrail
      Contact( "M0.4" )
      wire#w1
      Contact( "Auto" )
      wire#w3
      Coil( "DB05_SpoolCarriagePos".dbx0_2 )
   END_RUNG
   RUNG wire#powerrail
      Contact( "M1.3" )
      wire#w2
      Contact( "DB09_TablePos".dbx1_2 )
   END_RUNG wire#w1
   RUNG wire#powerrail
      Contact( "M3.2" )
   END_RUNG wire#w2
   RUNG wire#powerrail
      Contact( "M83.0" )
   END_RUNG wire#w1
   RUNG wire#powerrail
      Contact( "M83.1" )
   END_RUNG wire#w1
   RUNG wire#powerrail
      Contact( "V87_3" )
   END_RUNG wire#w1
   RUNG wire#powerrail
      Contact( "V87_4" )
   END_RUNG wire#w1
   RUNG wire#powerrail
      Contact( "DB80_Label".rotation )
   END_RUNG wire#w1
   RUNG wire#powerrail
      Contact( "DB80_Label".Step8 )
   END_RUNG wire#w1
   RUNG wire#powerrail
      Contact( "DB09_TablePos".dbx1_3 )
   END_RUNG wire#w3
   RUNG wire#powerrail
      Contact( "M32.4" )
      Contact( "DB09_TablePos".dbx1_2 )
      Contact( "M10.4" )
   END_RUNG wire#w3
   RUNG wire#powerrail
      Contact( "Manu" )
      Contact( "A11" )
      I_Contact( "DB22_DisplayData".dbx19_2 )
      I_Contact( "DB22_DisplayData".dbx19_3 )
      I_Contact( "DB22_DisplayData".dbx19_4 )
   END_RUNG wire#w3
   // the same network as SCL:
   "DB05_SpoolCarriagePos".dbx0_2 := (("M0.4" OR (("M1.3" OR "M3.2") AND "DB09_TablePos".dbx1_2) OR "M83.0" OR "M83.1" OR "V87_3" OR "V87_4" OR "DB80_Label".rotation OR "DB80_Label".Step8) AND "Auto") OR "DB09_TablePos".dbx1_3 OR ("M32.4" AND "DB09_TablePos".dbx1_2 AND "M10.4") OR ("Manu" AND "A11" AND NOT "DB22_DisplayData".dbx19_2 AND NOT "DB22_DisplayData".dbx19_3 AND NOT "DB22_DisplayData".dbx19_4);
END_REGION

REGION Network 21: Table rotation speed: Middle 2 for welder contrast
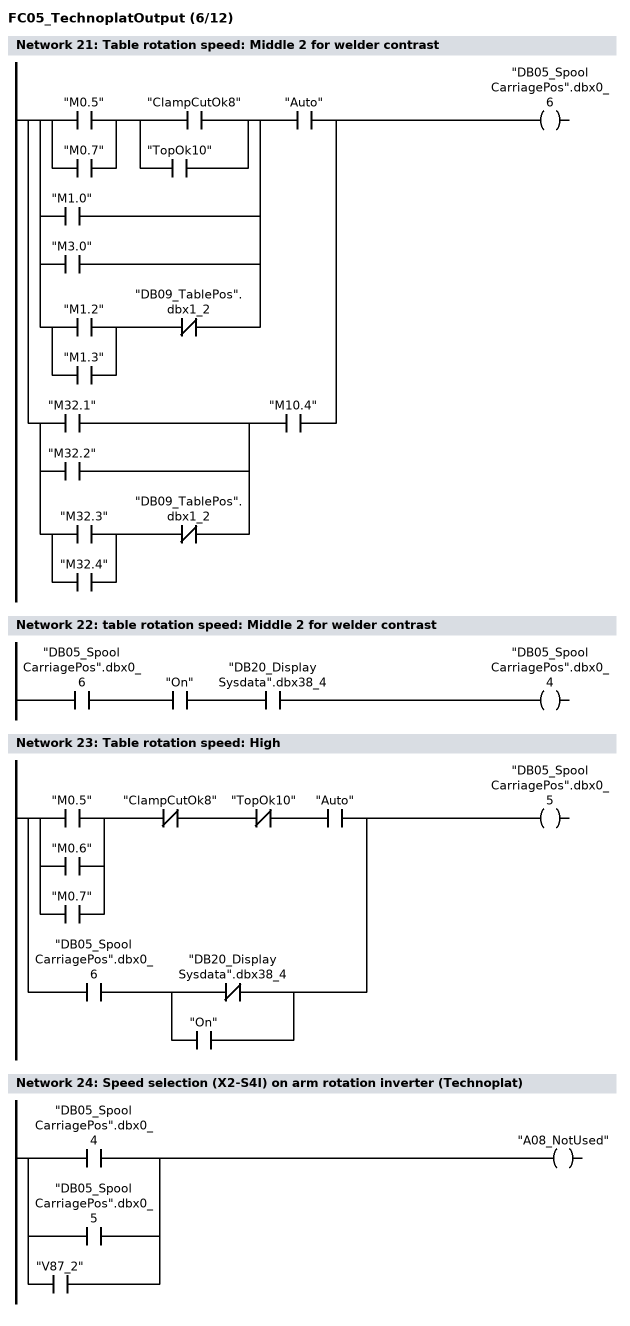
   RUNG wire#powerrail
      Contact( "M0.5" )
      wire#w1
      Contact( "ClampCutOk8" )
      wire#w2
      Contact( "Auto" )
      wire#w4
      Coil( "DB05_SpoolCarriagePos".dbx0_6 )
   END_RUNG
   RUNG wire#powerrail
      Contact( "M0.7" )
   END_RUNG wire#w1
   RUNG wire#w1
      Contact( "TopOk10" )
   END_RUNG wire#w2
   RUNG wire#powerrail
      Contact( "M1.0" )
   END_RUNG wire#w2
   RUNG wire#powerrail
      Contact( "M3.0" )
   END_RUNG wire#w2
   RUNG wire#powerrail
      Contact( "M1.2" )
      wire#w3
      I_Contact( "DB09_TablePos".dbx1_2 )
   END_RUNG wire#w2
   RUNG wire#powerrail
      Contact( "M1.3" )
   END_RUNG wire#w3
   RUNG wire#powerrail
      Contact( "M32.1" )
      wire#w5
      Contact( "M10.4" )
   END_RUNG wire#w4
   RUNG wire#powerrail
      Contact( "M32.2" )
   END_RUNG wire#w5
   RUNG wire#powerrail
      Contact( "M32.3" )
      wire#w6
      I_Contact( "DB09_TablePos".dbx1_2 )
   END_RUNG wire#w5
   RUNG wire#powerrail
      Contact( "M32.4" )
   END_RUNG wire#w6
   // the same network as SCL:
   "DB05_SpoolCarriagePos".dbx0_6 := (((("M0.5" OR "M0.7") AND ("ClampCutOk8" OR "TopOk10")) OR "M1.0" OR "M3.0" OR (("M1.2" OR "M1.3") AND NOT "DB09_TablePos".dbx1_2)) AND "Auto") OR (("M32.1" OR "M32.2" OR (("M32.3" OR "M32.4") AND NOT "DB09_TablePos".dbx1_2)) AND "M10.4");
END_REGION

REGION Network 22: table rotation speed: Middle 2 for welder contrast
   RUNG wire#powerrail
      Contact( "DB05_SpoolCarriagePos".dbx0_6 )
      Contact( "On" )
      Contact( "DB20_DisplaySysdata".dbx38_4 )
      Coil( "DB05_SpoolCarriagePos".dbx0_4 )
   END_RUNG
   // the same network as SCL:
   "DB05_SpoolCarriagePos".dbx0_4 := "DB05_SpoolCarriagePos".dbx0_6 AND "On" AND "DB20_DisplaySysdata".dbx38_4;
END_REGION

REGION Network 23: Table rotation speed: High
   RUNG wire#powerrail
      Contact( "M0.5" )
      wire#w1
      I_Contact( "ClampCutOk8" )
      I_Contact( "TopOk10" )
      Contact( "Auto" )
      wire#w2
      Coil( "DB05_SpoolCarriagePos".dbx0_5 )
   END_RUNG
   RUNG wire#powerrail
      Contact( "M0.6" )
   END_RUNG wire#w1
   RUNG wire#powerrail
      Contact( "M0.7" )
   END_RUNG wire#w1
   RUNG wire#powerrail
      Contact( "DB05_SpoolCarriagePos".dbx0_6 )
      wire#w3
      I_Contact( "DB20_DisplaySysdata".dbx38_4 )
   END_RUNG wire#w2
   RUNG wire#w3
      Contact( "On" )
   END_RUNG wire#w2
   // the same network as SCL:
   "DB05_SpoolCarriagePos".dbx0_5 := (("M0.5" OR "M0.6" OR "M0.7") AND NOT "ClampCutOk8" AND NOT "TopOk10" AND "Auto") OR ("DB05_SpoolCarriagePos".dbx0_6 AND (NOT "DB20_DisplaySysdata".dbx38_4 OR "On"));
END_REGION

REGION Network 24: Speed selection (X2-S4I) on arm rotation inverter (Technoplat)
   RUNG wire#powerrail
      Contact( "DB05_SpoolCarriagePos".dbx0_4 )
      wire#w1
      Coil( "A08_NotUsed" )
   END_RUNG
   RUNG wire#powerrail
      Contact( "DB05_SpoolCarriagePos".dbx0_5 )
   END_RUNG wire#w1
   RUNG wire#powerrail
      Contact( "V87_2" )
   END_RUNG wire#w1
   // the same network as SCL:
   "A08_NotUsed" := "DB05_SpoolCarriagePos".dbx0_4 OR "DB05_SpoolCarriagePos".dbx0_5 OR "V87_2";
END_REGION

REGION Network 25: SPARE - Speed selection (X3-S5I) on arm rotation inverter (Techn
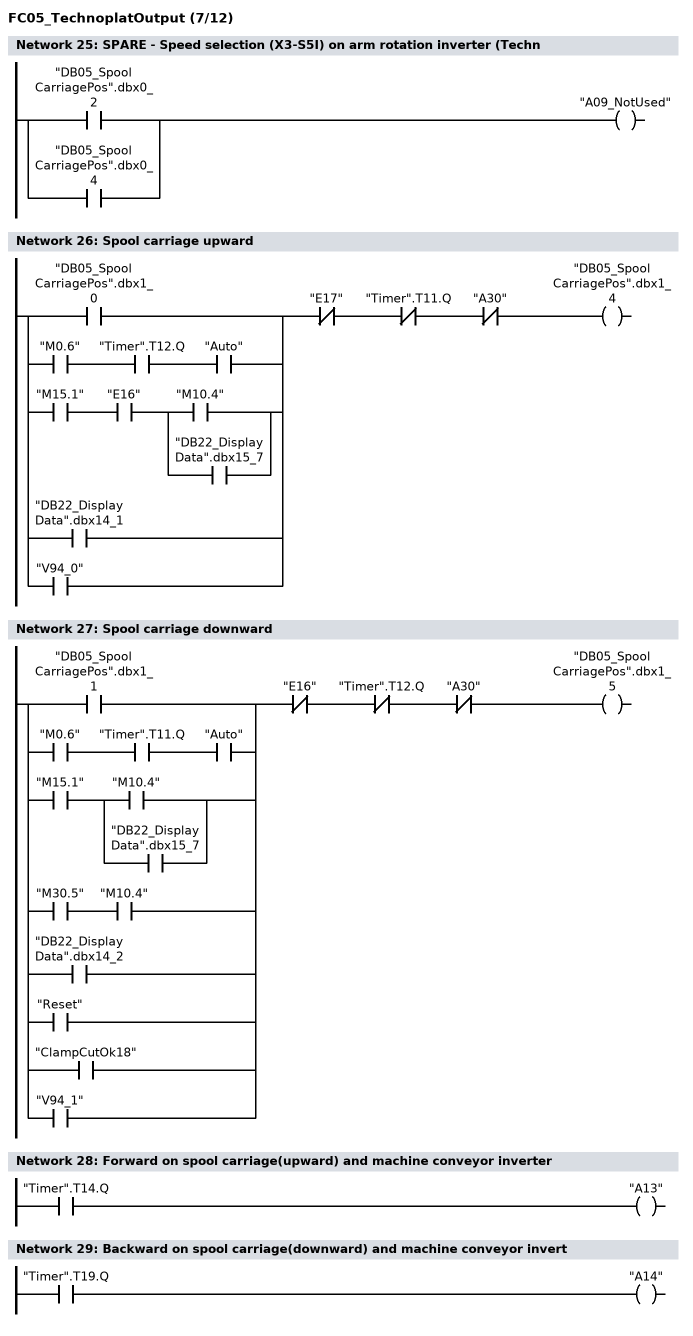
   RUNG wire#powerrail
      Contact( "DB05_SpoolCarriagePos".dbx0_2 )
      wire#w1
      Coil( "A09_NotUsed" )
   END_RUNG
   RUNG wire#powerrail
      Contact( "DB05_SpoolCarriagePos".dbx0_4 )
   END_RUNG wire#w1
   // the same network as SCL:
   "A09_NotUsed" := "DB05_SpoolCarriagePos".dbx0_2 OR "DB05_SpoolCarriagePos".dbx0_4;
END_REGION

REGION Network 26: Spool carriage upward
   RUNG wire#powerrail
      Contact( "DB05_SpoolCarriagePos".dbx1_0 )
      wire#w1
      I_Contact( "E17" )
      I_Contact( "Timer".T11.Q )
      I_Contact( "A30" )
      Coil( "DB05_SpoolCarriagePos".dbx1_4 )
   END_RUNG
   RUNG wire#powerrail
      Contact( "M0.6" )
      Contact( "Timer".T12.Q )
      Contact( "Auto" )
   END_RUNG wire#w1
   RUNG wire#powerrail
      Contact( "M15.1" )
      Contact( "E16" )
      wire#w2
      Contact( "M10.4" )
   END_RUNG wire#w1
   RUNG wire#w2
      Contact( "DB22_DisplayData".dbx15_7 )
   END_RUNG wire#w1
   RUNG wire#powerrail
      Contact( "DB22_DisplayData".dbx14_1 )
   END_RUNG wire#w1
   RUNG wire#powerrail
      Contact( "V94_0" )
   END_RUNG wire#w1
   // the same network as SCL:
   "DB05_SpoolCarriagePos".dbx1_4 := ("DB05_SpoolCarriagePos".dbx1_0 OR ("M0.6" AND "Timer".T12.Q AND "Auto") OR ("M15.1" AND "E16" AND ("M10.4" OR "DB22_DisplayData".dbx15_7)) OR "DB22_DisplayData".dbx14_1 OR "V94_0") AND NOT "E17" AND NOT "Timer".T11.Q AND NOT "A30";
END_REGION

REGION Network 27: Spool carriage downward
   RUNG wire#powerrail
      Contact( "DB05_SpoolCarriagePos".dbx1_1 )
      wire#w1
      I_Contact( "E16" )
      I_Contact( "Timer".T12.Q )
      I_Contact( "A30" )
      Coil( "DB05_SpoolCarriagePos".dbx1_5 )
   END_RUNG
   RUNG wire#powerrail
      Contact( "M0.6" )
      Contact( "Timer".T11.Q )
      Contact( "Auto" )
   END_RUNG wire#w1
   RUNG wire#powerrail
      Contact( "M15.1" )
      wire#w2
      Contact( "M10.4" )
   END_RUNG wire#w1
   RUNG wire#w2
      Contact( "DB22_DisplayData".dbx15_7 )
   END_RUNG wire#w1
   RUNG wire#powerrail
      Contact( "M30.5" )
      Contact( "M10.4" )
   END_RUNG wire#w1
   RUNG wire#powerrail
      Contact( "DB22_DisplayData".dbx14_2 )
   END_RUNG wire#w1
   RUNG wire#powerrail
      Contact( "Reset" )
   END_RUNG wire#w1
   RUNG wire#powerrail
      Contact( "ClampCutOk18" )
   END_RUNG wire#w1
   RUNG wire#powerrail
      Contact( "V94_1" )
   END_RUNG wire#w1
   // the same network as SCL:
   "DB05_SpoolCarriagePos".dbx1_5 := ("DB05_SpoolCarriagePos".dbx1_1 OR ("M0.6" AND "Timer".T11.Q AND "Auto") OR ("M15.1" AND ("M10.4" OR "DB22_DisplayData".dbx15_7)) OR ("M30.5" AND "M10.4") OR "DB22_DisplayData".dbx14_2 OR "Reset" OR "ClampCutOk18" OR "V94_1") AND NOT "E16" AND NOT "Timer".T12.Q AND NOT "A30";
END_REGION

REGION Network 28: Forward on spool carriage(upward) and machine conveyor inverter
   RUNG wire#powerrail
      Contact( "Timer".T14.Q )
      Coil( "A13" )
   END_RUNG
   // the same network as SCL:
   "A13" := "Timer".T14.Q;
END_REGION

REGION Network 29: Backward on spool carriage(downward) and machine conveyor invert
   RUNG wire#powerrail
      Contact( "Timer".T19.Q )
      Coil( "A14" )
   END_RUNG
   // the same network as SCL:
   "A14" := "Timer".T19.Q;
END_REGION

REGION Network 30: Motor for spool carriage (Helix)
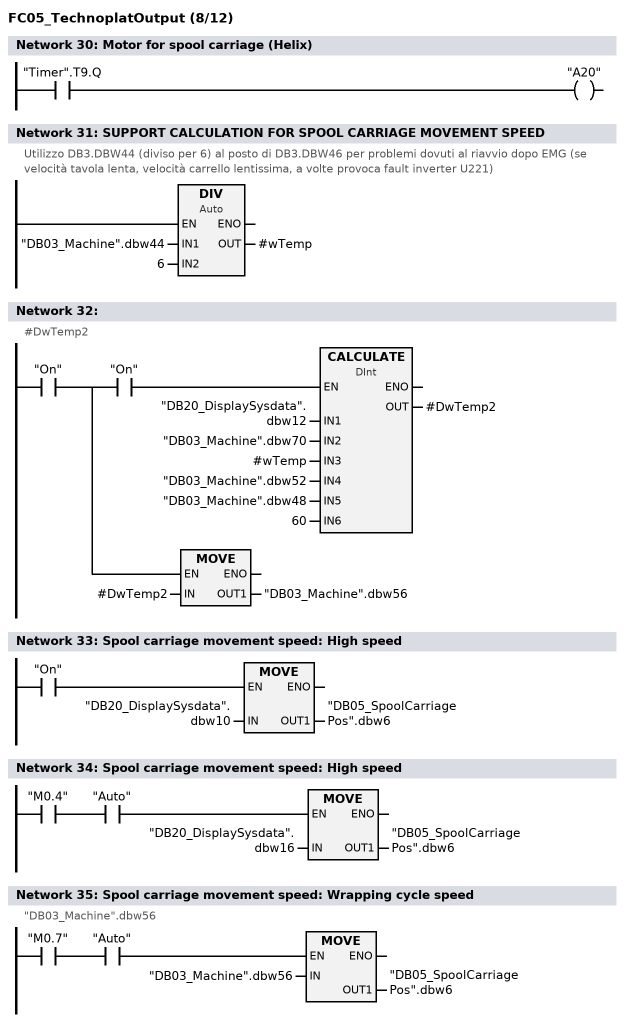
   RUNG wire#powerrail
      Contact( "Timer".T9.Q )
      Coil( "A20" )
   END_RUNG
   // the same network as SCL:
   "A20" := "Timer".T9.Q;
END_REGION

REGION Network 31: SUPPORT CALCULATION FOR SPOOL CARRIAGE MOVEMENT SPEED
   // Utilizzo DB3.DBW44 (diviso per 6) al posto di DB3.DBW46 per problemi dovuti al riavvio dopo EMG (se velocità tavola lenta, velocità carrello lentissima, a volte provoca fault inverter U221)
   RUNG wire#powerrail
      Div(in1 := "DB03_Machine".dbw44, in2 := 6, out => #wTemp)
   END_RUNG
   // the same network as SCL:
   #wTemp := "DB03_Machine".dbw44 / 6;
END_REGION

REGION Network 32
   // #DwTemp2
   RUNG wire#powerrail
      Contact( "On" )
      wire#w1
      Contact( "On" )
      { S7_Templates := "SrcType := DInt"; S7_GenerateENO := "TRUE"; S7_Expression := "((In1-In2)*In3*In4)/(In5*In6)" } Calculate(in1 := "DB20_DisplaySysdata".dbw12, in2 := "DB03_Machine".dbw70, in3 := #wTemp, in4 := "DB03_Machine".dbw52, in5 := "DB03_Machine".dbw48, in6 := 60, out => #DwTemp2)
   END_RUNG
   RUNG wire#w1
      { S7_GenerateENO := "TRUE" } Move(in := #DwTemp2, out1 => "DB03_Machine".dbw56)
   END_RUNG
   // the same network as SCL:
   IF "On" AND "On" THEN
       #DwTemp2 := (("DB20_DisplaySysdata".dbw12-"DB03_Machine".dbw70)*#wTemp*"DB03_Machine".dbw52)/("DB03_Machine".dbw48*60);
   END_IF;
   IF "On" THEN "DB03_Machine".dbw56 := #DwTemp2; END_IF;
END_REGION

REGION Network 33: Spool carriage movement speed: High speed
   RUNG wire#powerrail
      Contact( "On" )
      { S7_GenerateENO := "TRUE" } Move(in := "DB20_DisplaySysdata".dbw10, out1 => "DB05_SpoolCarriagePos".dbw6)
   END_RUNG
   // the same network as SCL:
   IF "On" THEN "DB05_SpoolCarriagePos".dbw6 := "DB20_DisplaySysdata".dbw10; END_IF;
END_REGION

REGION Network 34: Spool carriage movement speed: High speed
   RUNG wire#powerrail
      Contact( "M0.4" )
      Contact( "Auto" )
      { S7_GenerateENO := "TRUE" } Move(in := "DB20_DisplaySysdata".dbw16, out1 => "DB05_SpoolCarriagePos".dbw6)
   END_RUNG
   // the same network as SCL:
   IF "M0.4" AND "Auto" THEN "DB05_SpoolCarriagePos".dbw6 := "DB20_DisplaySysdata".dbw16; END_IF;
END_REGION

REGION Network 35: Spool carriage movement speed: Wrapping cycle speed
   // "DB03_Machine".dbw56
   RUNG wire#powerrail
      Contact( "M0.7" )
      Contact( "Auto" )
      { S7_GenerateENO := "TRUE" } Move(in := "DB03_Machine".dbw56, out1 => "DB05_SpoolCarriagePos".dbw6)
   END_RUNG
   // the same network as SCL:
   IF "M0.7" AND "Auto" THEN "DB05_SpoolCarriagePos".dbw6 := "DB03_Machine".dbw56; END_IF;
END_REGION

REGION Network 36: Spool carriage movement speed: Low speed
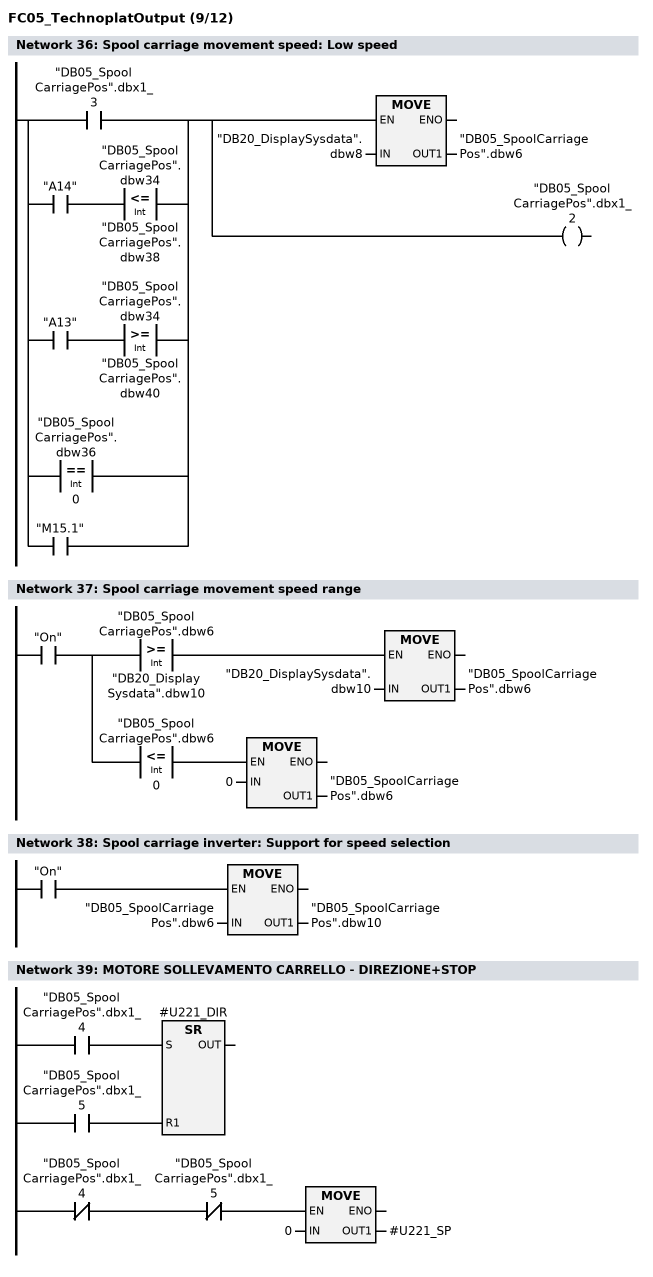
   RUNG wire#powerrail
      Contact( "DB05_SpoolCarriagePos".dbx1_3 )
      wire#w1
      { S7_GenerateENO := "TRUE" } Move(in := "DB20_DisplaySysdata".dbw8, out1 => "DB05_SpoolCarriagePos".dbw6)
   END_RUNG
   RUNG wire#powerrail
      Contact( "A14" )
      { S7_Templates := "SrcType := Int" } LE_Contact(in1 := "DB05_SpoolCarriagePos".dbw34, in2 := "DB05_SpoolCarriagePos".dbw38)
   END_RUNG wire#w1
   RUNG wire#powerrail
      Contact( "A13" )
      { S7_Templates := "SrcType := Int" } GE_Contact(in1 := "DB05_SpoolCarriagePos".dbw34, in2 := "DB05_SpoolCarriagePos".dbw40)
   END_RUNG wire#w1
   RUNG wire#powerrail
      { S7_Templates := "SrcType := Int" } EQ_Contact(in1 := "DB05_SpoolCarriagePos".dbw36, in2 := 0)
   END_RUNG wire#w1
   RUNG wire#powerrail
      Contact( "M15.1" )
   END_RUNG wire#w1
   RUNG wire#w1
      Coil( "DB05_SpoolCarriagePos".dbx1_2 )
   END_RUNG
   // the same network as SCL:
   #_w1 := "DB05_SpoolCarriagePos".dbx1_3 OR ("A14" AND ("DB05_SpoolCarriagePos".dbw34 <= "DB05_SpoolCarriagePos".dbw38)) OR ("A13" AND ("DB05_SpoolCarriagePos".dbw34 >= "DB05_SpoolCarriagePos".dbw40)) OR ("DB05_SpoolCarriagePos".dbw36 = 0) OR "M15.1";
   IF #_w1 THEN "DB05_SpoolCarriagePos".dbw6 := "DB20_DisplaySysdata".dbw8; END_IF;
   "DB05_SpoolCarriagePos".dbx1_2 := #_w1;
END_REGION

REGION Network 37: Spool carriage movement speed range
   RUNG wire#powerrail
      Contact( "On" )
      wire#w1
      { S7_Templates := "SrcType := Int" } GE_Contact(in1 := "DB05_SpoolCarriagePos".dbw6, in2 := "DB20_DisplaySysdata".dbw10)
      { S7_GenerateENO := "TRUE" } Move(in := "DB20_DisplaySysdata".dbw10, out1 => "DB05_SpoolCarriagePos".dbw6)
   END_RUNG
   RUNG wire#w1
      { S7_Templates := "SrcType := Int" } LE_Contact(in1 := "DB05_SpoolCarriagePos".dbw6, in2 := 0)
      { S7_GenerateENO := "TRUE" } Move(in := 0, out1 => "DB05_SpoolCarriagePos".dbw6)
   END_RUNG
   // the same network as SCL:
   IF "On" AND ("DB05_SpoolCarriagePos".dbw6 >= "DB20_DisplaySysdata".dbw10) THEN
       "DB05_SpoolCarriagePos".dbw6 := "DB20_DisplaySysdata".dbw10;
   END_IF;
   IF "On" AND ("DB05_SpoolCarriagePos".dbw6 <= 0) THEN "DB05_SpoolCarriagePos".dbw6 := 0; END_IF;
END_REGION

REGION Network 38: Spool carriage inverter: Support for speed selection
   RUNG wire#powerrail
      Contact( "On" )
      { S7_GenerateENO := "TRUE" } Move(in := "DB05_SpoolCarriagePos".dbw6, out1 => "DB05_SpoolCarriagePos".dbw10)
   END_RUNG
   // the same network as SCL:
   IF "On" THEN "DB05_SpoolCarriagePos".dbw10 := "DB05_SpoolCarriagePos".dbw6; END_IF;
END_REGION

REGION Network 39: MOTORE SOLLEVAMENTO CARRELLO - DIREZIONE+STOP
   RUNG wire#powerrail
      Contact( "DB05_SpoolCarriagePos".dbx1_4 )
      S_SR(operand := #U221_DIR, r1 := wire#w1)
   END_RUNG
   RUNG wire#powerrail
      Contact( "DB05_SpoolCarriagePos".dbx1_5 )
   END_RUNG wire#w1
   RUNG wire#powerrail
      I_Contact( "DB05_SpoolCarriagePos".dbx1_4 )
      I_Contact( "DB05_SpoolCarriagePos".dbx1_5 )
      Move(in := 0, out1 => #U221_SP)
   END_RUNG
   // the same network as SCL:
   IF "DB05_SpoolCarriagePos".dbx1_4 THEN
       #U221_DIR := TRUE;   // SR flip-flop
   END_IF;
   IF "DB05_SpoolCarriagePos".dbx1_5 THEN #U221_DIR := FALSE; END_IF;
   IF NOT "DB05_SpoolCarriagePos".dbx1_4 AND NOT "DB05_SpoolCarriagePos".dbx1_5 THEN #U221_SP := 0; END_IF;
END_REGION

REGION Network 40: MOTORE SOLLEVAMENTO CARRELLO - RIF.VELOCITA' + START
   // 2250 RPM = 75 HZ = 100% (3000@100HZ)
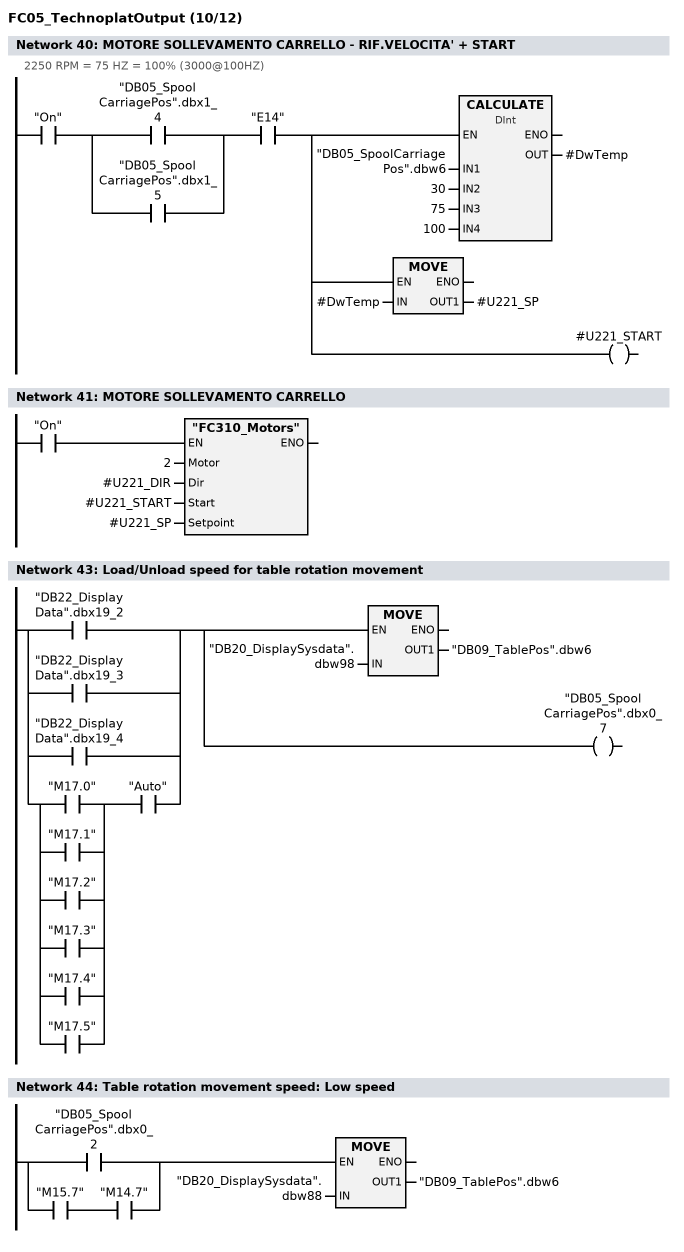
   RUNG wire#powerrail
      Contact( "On" )
      wire#w1
      Contact( "DB05_SpoolCarriagePos".dbx1_4 )
      wire#w2
      Contact( "E14" )
      wire#w3
      { S7_Templates := "SrcType := DInt"; S7_Expression := "(IN1*IN2*IN3)/IN4" } Calculate(in1 := "DB05_SpoolCarriagePos".dbw6, in2 := 30, in3 := 75, in4 := 100, out => #DwTemp)
   END_RUNG
   RUNG wire#w1
      Contact( "DB05_SpoolCarriagePos".dbx1_5 )
   END_RUNG wire#w2
   RUNG wire#w3
      Move(in := #DwTemp, out1 => #U221_SP)
   END_RUNG
   RUNG wire#w3
      Coil( #U221_START )
   END_RUNG
   // the same network as SCL:
   #_w1 := "On" AND ("DB05_SpoolCarriagePos".dbx1_4 OR "DB05_SpoolCarriagePos".dbx1_5) AND "E14";
   IF #_w1 THEN
       #DwTemp := ("DB05_SpoolCarriagePos".dbw6*30*75)/100;
       #U221_SP := #DwTemp;
   END_IF;
   #U221_START := #_w1;
END_REGION

REGION Network 41: MOTORE SOLLEVAMENTO CARRELLO
   RUNG wire#powerrail
      Contact( "On" )
      "FC310_Motors"(Motor := 2, Dir := #U221_DIR, Start := #U221_START, Setpoint := #U221_SP)
   END_RUNG
   // the same network as SCL:
   IF "On" THEN
       "FC310_Motors"(Motor := 2, Dir := #U221_DIR, Start := #U221_START, Setpoint := #U221_SP);
   END_IF;
END_REGION

REGION Network 42: Carriage and arm rotation speed conversion
END_REGION

REGION Network 43: Load/Unload speed for table rotation movement
   RUNG wire#powerrail
      Contact( "DB22_DisplayData".dbx19_2 )
      wire#w1
      { S7_GenerateENO := "TRUE" } Move(in := "DB20_DisplaySysdata".dbw98, out1 => "DB09_TablePos".dbw6)
   END_RUNG
   RUNG wire#powerrail
      Contact( "DB22_DisplayData".dbx19_3 )
   END_RUNG wire#w1
   RUNG wire#powerrail
      Contact( "DB22_DisplayData".dbx19_4 )
   END_RUNG wire#w1
   RUNG wire#powerrail
      Contact( "M17.0" )
      wire#w2
      Contact( "Auto" )
   END_RUNG wire#w1
   RUNG wire#powerrail
      Contact( "M17.1" )
   END_RUNG wire#w2
   RUNG wire#powerrail
      Contact( "M17.2" )
   END_RUNG wire#w2
   RUNG wire#powerrail
      Contact( "M17.3" )
   END_RUNG wire#w2
   RUNG wire#powerrail
      Contact( "M17.4" )
   END_RUNG wire#w2
   RUNG wire#powerrail
      Contact( "M17.5" )
   END_RUNG wire#w2
   RUNG wire#w1
      Coil( "DB05_SpoolCarriagePos".dbx0_7 )
   END_RUNG
   // the same network as SCL:
   #_w1 := "DB22_DisplayData".dbx19_2 OR "DB22_DisplayData".dbx19_3 OR "DB22_DisplayData".dbx19_4 OR (("M17.0" OR "M17.1" OR "M17.2" OR "M17.3" OR "M17.4" OR "M17.5") AND "Auto");
   IF #_w1 THEN "DB09_TablePos".dbw6 := "DB20_DisplaySysdata".dbw98; END_IF;
   "DB05_SpoolCarriagePos".dbx0_7 := #_w1;
END_REGION

REGION Network 44: Table rotation movement speed: Low speed
   RUNG wire#powerrail
      Contact( "DB05_SpoolCarriagePos".dbx0_2 )
      wire#w1
      { S7_GenerateENO := "TRUE" } Move(in := "DB20_DisplaySysdata".dbw88, out1 => "DB09_TablePos".dbw6)
   END_RUNG
   RUNG wire#powerrail
      Contact( "M15.7" )
      Contact( "M14.7" )
   END_RUNG wire#w1
   // the same network as SCL:
   IF "DB05_SpoolCarriagePos".dbx0_2 OR ("M15.7" AND "M14.7") THEN
       "DB09_TablePos".dbw6 := "DB20_DisplaySysdata".dbw88;
   END_IF;
END_REGION

REGION Network 45: EXTRA LOW
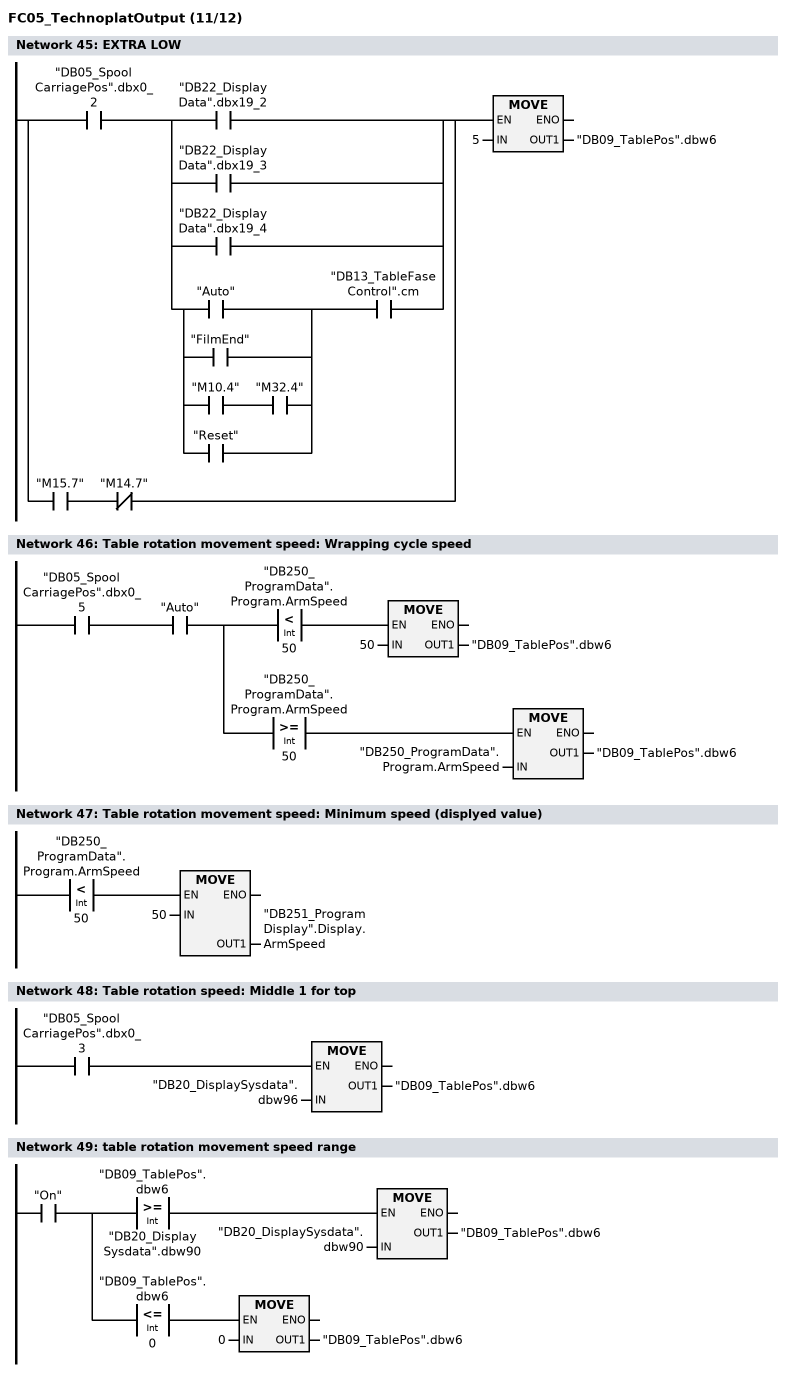
   RUNG wire#powerrail
      Contact( "DB05_SpoolCarriagePos".dbx0_2 )
      wire#w1
      Contact( "DB22_DisplayData".dbx19_2 )
      wire#w2
      { S7_GenerateENO := "TRUE" } Move(in := 5, out1 => "DB09_TablePos".dbw6)
   END_RUNG
   RUNG wire#w1
      Contact( "DB22_DisplayData".dbx19_3 )
   END_RUNG wire#w2
   RUNG wire#w1
      Contact( "DB22_DisplayData".dbx19_4 )
   END_RUNG wire#w2
   RUNG wire#w1
      Contact( "Auto" )
      wire#w3
      Contact( "DB13_TableFaseControl".cm )
   END_RUNG wire#w2
   RUNG wire#w1
      Contact( "FilmEnd" )
   END_RUNG wire#w3
   RUNG wire#w1
      Contact( "M10.4" )
      Contact( "M32.4" )
   END_RUNG wire#w3
   RUNG wire#w1
      Contact( "Reset" )
   END_RUNG wire#w3
   RUNG wire#powerrail
      Contact( "M15.7" )
      I_Contact( "M14.7" )
   END_RUNG wire#w2
   // the same network as SCL:
   IF ("DB05_SpoolCarriagePos".dbx0_2 AND ("DB22_DisplayData".dbx19_2 OR "DB22_DisplayData".dbx19_3 OR "DB22_DisplayData".dbx19_4 OR (("Auto" OR "FilmEnd" OR ("M10.4" AND "M32.4") OR "Reset") AND "DB13_TableFaseControl".cm))) OR ("M15.7" AND NOT "M14.7") THEN
       "DB09_TablePos".dbw6 := 5;
   END_IF;
END_REGION

REGION Network 46: Table rotation movement speed: Wrapping cycle speed
   RUNG wire#powerrail
      Contact( "DB05_SpoolCarriagePos".dbx0_5 )
      Contact( "Auto" )
      wire#w1
      { S7_Templates := "SrcType := Int" } LT_Contact(in1 := "DB250_ProgramData".Program.ArmSpeed, in2 := 50)
      { S7_GenerateENO := "TRUE" } Move(in := 50, out1 => "DB09_TablePos".dbw6)
   END_RUNG
   RUNG wire#w1
      { S7_Templates := "SrcType := Int" } GE_Contact(in1 := "DB250_ProgramData".Program.ArmSpeed, in2 := 50)
      { S7_GenerateENO := "TRUE" } Move(in := "DB250_ProgramData".Program.ArmSpeed, out1 => "DB09_TablePos".dbw6)
   END_RUNG
   // the same network as SCL:
   #_w1 := "DB05_SpoolCarriagePos".dbx0_5 AND "Auto";
   IF #_w1 AND ("DB250_ProgramData".Program.ArmSpeed < 50) THEN "DB09_TablePos".dbw6 := 50; END_IF;
   IF #_w1 AND ("DB250_ProgramData".Program.ArmSpeed >= 50) THEN
       "DB09_TablePos".dbw6 := "DB250_ProgramData".Program.ArmSpeed;
   END_IF;
END_REGION

REGION Network 47: Table rotation movement speed: Minimum speed (displyed value)
   RUNG wire#powerrail
      { S7_Templates := "SrcType := Int" } LT_Contact(in1 := "DB250_ProgramData".Program.ArmSpeed, in2 := 50)
      { S7_GenerateENO := "TRUE" } Move(in := 50, out1 => "DB251_ProgramDisplay".Display.ArmSpeed)
   END_RUNG
   // the same network as SCL:
   IF "DB250_ProgramData".Program.ArmSpeed < 50 THEN "DB251_ProgramDisplay".Display.ArmSpeed := 50; END_IF;
END_REGION

REGION Network 48: Table rotation speed: Middle 1 for top
   RUNG wire#powerrail
      Contact( "DB05_SpoolCarriagePos".dbx0_3 )
      { S7_GenerateENO := "TRUE" } Move(in := "DB20_DisplaySysdata".dbw96, out1 => "DB09_TablePos".dbw6)
   END_RUNG
   // the same network as SCL:
   IF "DB05_SpoolCarriagePos".dbx0_3 THEN "DB09_TablePos".dbw6 := "DB20_DisplaySysdata".dbw96; END_IF;
END_REGION

REGION Network 49: table rotation movement speed range
   RUNG wire#powerrail
      Contact( "On" )
      wire#w1
      { S7_Templates := "SrcType := Int" } GE_Contact(in1 := "DB09_TablePos".dbw6, in2 := "DB20_DisplaySysdata".dbw90)
      { S7_GenerateENO := "TRUE" } Move(in := "DB20_DisplaySysdata".dbw90, out1 => "DB09_TablePos".dbw6)
   END_RUNG
   RUNG wire#w1
      { S7_Templates := "SrcType := Int" } LE_Contact(in1 := "DB09_TablePos".dbw6, in2 := 0)
      { S7_GenerateENO := "TRUE" } Move(in := 0, out1 => "DB09_TablePos".dbw6)
   END_RUNG
   // the same network as SCL:
   IF "On" AND ("DB09_TablePos".dbw6 >= "DB20_DisplaySysdata".dbw90) THEN
       "DB09_TablePos".dbw6 := "DB20_DisplaySysdata".dbw90;
   END_IF;
   IF "On" AND ("DB09_TablePos".dbw6 <= 0) THEN "DB09_TablePos".dbw6 := 0; END_IF;
END_REGION

REGION Network 50: table rotation inverter: Support for speed selection
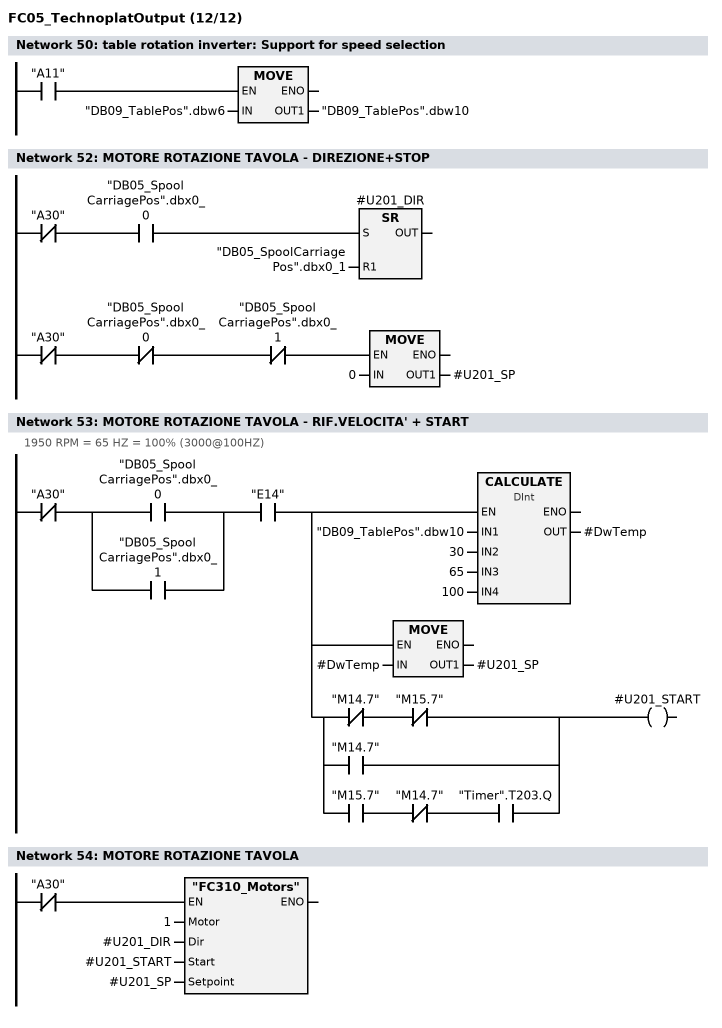
   RUNG wire#powerrail
      Contact( "A11" )
      { S7_GenerateENO := "TRUE" } Move(in := "DB09_TablePos".dbw6, out1 => "DB09_TablePos".dbw10)
   END_RUNG
   // the same network as SCL:
   IF "A11" THEN "DB09_TablePos".dbw10 := "DB09_TablePos".dbw6; END_IF;
END_REGION

REGION Network 51: Table rotation speed conversion
END_REGION

REGION Network 52: MOTORE ROTAZIONE TAVOLA - DIREZIONE+STOP
   RUNG wire#powerrail
      I_Contact( "A30" )
      Contact( "DB05_SpoolCarriagePos".dbx0_0 )
      S_SR(operand := #U201_DIR, r1 := "DB05_SpoolCarriagePos".dbx0_1)
   END_RUNG
   RUNG wire#powerrail
      I_Contact( "A30" )
      I_Contact( "DB05_SpoolCarriagePos".dbx0_0 )
      I_Contact( "DB05_SpoolCarriagePos".dbx0_1 )
      Move(in := 0, out1 => #U201_SP)
   END_RUNG
   // the same network as SCL:
   IF NOT "A30" AND "DB05_SpoolCarriagePos".dbx0_0 THEN
       #U201_DIR := TRUE;   // SR flip-flop
   END_IF;
   IF "DB05_SpoolCarriagePos".dbx0_1 THEN #U201_DIR := FALSE; END_IF;
   IF NOT "A30" AND NOT "DB05_SpoolCarriagePos".dbx0_0 AND NOT "DB05_SpoolCarriagePos".dbx0_1 THEN
       #U201_SP := 0;
   END_IF;
END_REGION

REGION Network 53: MOTORE ROTAZIONE TAVOLA - RIF.VELOCITA' + START
   // 1950 RPM = 65 HZ = 100% (3000@100HZ)
   RUNG wire#powerrail
      I_Contact( "A30" )
      wire#w1
      Contact( "DB05_SpoolCarriagePos".dbx0_0 )
      wire#w2
      Contact( "E14" )
      wire#w3
      { S7_Templates := "SrcType := DInt"; S7_Expression := "(IN1*IN2*IN3)/IN4" } Calculate(in1 := "DB09_TablePos".dbw10, in2 := 30, in3 := 65, in4 := 100, out => #DwTemp)
   END_RUNG
   RUNG wire#w1
      Contact( "DB05_SpoolCarriagePos".dbx0_1 )
   END_RUNG wire#w2
   RUNG wire#w3
      Move(in := #DwTemp, out1 => #U201_SP)
   END_RUNG
   RUNG wire#w3
      I_Contact( "M14.7" )
      I_Contact( "M15.7" )
      wire#w4
      Coil( #U201_START )
   END_RUNG
   RUNG wire#w3
      Contact( "M14.7" )
   END_RUNG wire#w4
   RUNG wire#w3
      Contact( "M15.7" )
      I_Contact( "M14.7" )
      Contact( "Timer".T203.Q )
   END_RUNG wire#w4
   // the same network as SCL:
   #_w1 := NOT "A30" AND ("DB05_SpoolCarriagePos".dbx0_0 OR "DB05_SpoolCarriagePos".dbx0_1) AND "E14";
   IF #_w1 THEN
       #DwTemp := ("DB09_TablePos".dbw10*30*65)/100;
       #U201_SP := #DwTemp;
   END_IF;
   #U201_START := #_w1 AND ((NOT "M14.7" AND NOT "M15.7") OR "M14.7" OR ("M15.7" AND NOT "M14.7" AND "Timer".T203.Q));
END_REGION

REGION Network 54: MOTORE ROTAZIONE TAVOLA
   RUNG wire#powerrail
      I_Contact( "A30" )
      "FC310_Motors"(Motor := 1, Dir := #U201_DIR, Start := #U201_START, Setpoint := #U201_SP)
   END_RUNG
   // the same network as SCL:
   IF NOT "A30" THEN
       "FC310_Motors"(Motor := 1, Dir := #U201_DIR, Start := #U201_START, Setpoint := #U201_SP);
   END_IF;
END_REGION
END_FUNCTION

FUNCTION "FC04_TechnoplatAlarm" : Void   // FC4, LAD
TITLE = Alarm for the machine
{ S7_Optimized_Access := 'FALSE' }
AUTHOR : Robopac
VERSION : 0.0
// stored: AutoNumber false, IsIECCheckEnabled false, SetENOAutomatically false, UDAEnableTagReadback false
BEGIN

REGION Network 1: Alarm 1: Pressure switch (Technoplat)
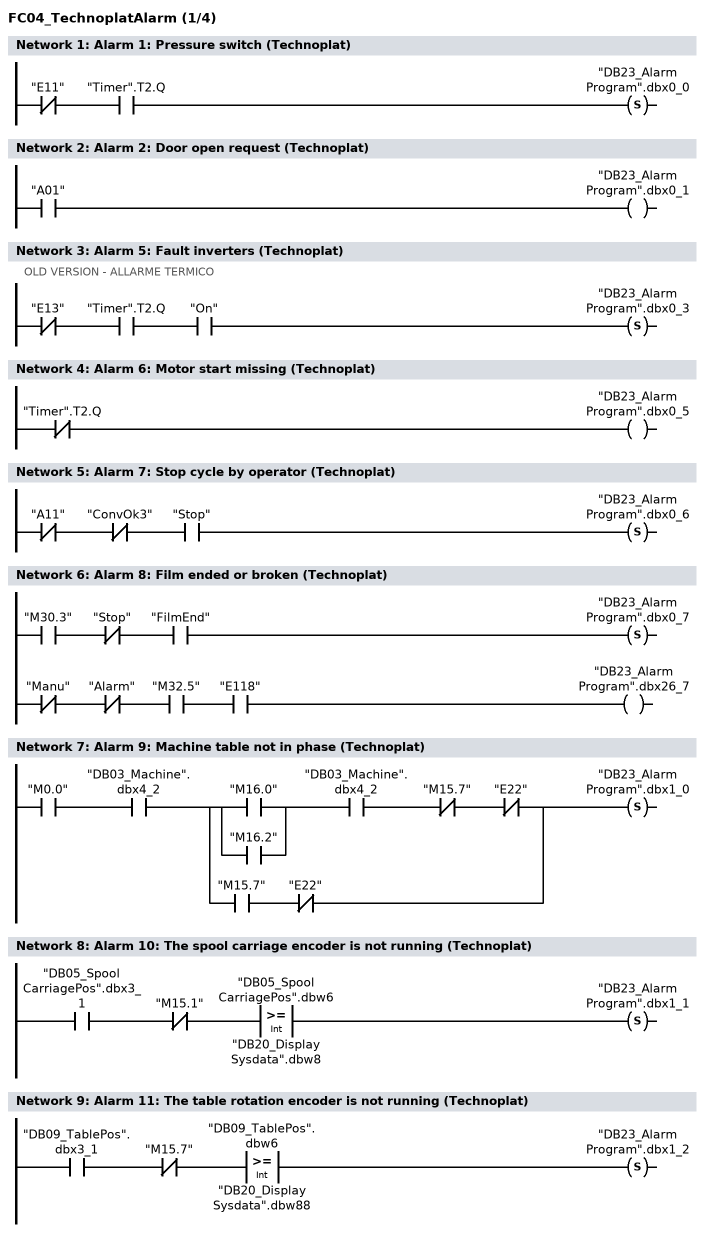
   RUNG wire#powerrail
      I_Contact( "E11" )
      Contact( "Timer".T2.Q )
      S_Coil( "DB23_AlarmProgram".dbx0_0 )
   END_RUNG
   // the same network as SCL:
   IF NOT "E11" AND "Timer".T2.Q THEN "DB23_AlarmProgram".dbx0_0 := TRUE; END_IF;
END_REGION

REGION Network 2: Alarm 2: Door open request (Technoplat)
   RUNG wire#powerrail
      Contact( "A01" )
      Coil( "DB23_AlarmProgram".dbx0_1 )
   END_RUNG
   // the same network as SCL:
   "DB23_AlarmProgram".dbx0_1 := "A01";
END_REGION

REGION Network 3: Alarm 5: Fault inverters (Technoplat)
   // OLD VERSION - ALLARME TERMICO
   RUNG wire#powerrail
      I_Contact( "E13" )
      Contact( "Timer".T2.Q )
      Contact( "On" )
      S_Coil( "DB23_AlarmProgram".dbx0_3 )
   END_RUNG
   // the same network as SCL:
   IF NOT "E13" AND "Timer".T2.Q AND "On" THEN "DB23_AlarmProgram".dbx0_3 := TRUE; END_IF;
END_REGION

REGION Network 4: Alarm 6: Motor start missing (Technoplat)
   RUNG wire#powerrail
      I_Contact( "Timer".T2.Q )
      Coil( "DB23_AlarmProgram".dbx0_5 )
   END_RUNG
   // the same network as SCL:
   "DB23_AlarmProgram".dbx0_5 := NOT "Timer".T2.Q;
END_REGION

REGION Network 5: Alarm 7: Stop cycle by operator (Technoplat)
   RUNG wire#powerrail
      I_Contact( "A11" )
      I_Contact( "ConvOk3" )
      Contact( "Stop" )
      S_Coil( "DB23_AlarmProgram".dbx0_6 )
   END_RUNG
   // the same network as SCL:
   IF NOT "A11" AND NOT "ConvOk3" AND "Stop" THEN "DB23_AlarmProgram".dbx0_6 := TRUE; END_IF;
END_REGION

REGION Network 6: Alarm 8: Film ended or broken (Technoplat)
   RUNG wire#powerrail
      Contact( "M30.3" )
      I_Contact( "Stop" )
      Contact( "FilmEnd" )
      S_Coil( "DB23_AlarmProgram".dbx0_7 )
   END_RUNG
   RUNG wire#powerrail
      I_Contact( "Manu" )
      I_Contact( "Alarm" )
      Contact( "M32.5" )
      Contact( "E118" )
      Coil( "DB23_AlarmProgram".dbx26_7 )
   END_RUNG
   // the same network as SCL:
   IF "M30.3" AND NOT "Stop" AND "FilmEnd" THEN "DB23_AlarmProgram".dbx0_7 := TRUE; END_IF;
   "DB23_AlarmProgram".dbx26_7 := NOT "Manu" AND NOT "Alarm" AND "M32.5" AND "E118";
END_REGION

REGION Network 7: Alarm 9: Machine table not in phase (Technoplat)
   RUNG wire#powerrail
      Contact( "M0.0" )
      Contact( "DB03_Machine".dbx4_2 )
      wire#w1
      Contact( "M16.0" )
      wire#w2
      Contact( "DB03_Machine".dbx4_2 )
      I_Contact( "M15.7" )
      I_Contact( "E22" )
      wire#w3
      S_Coil( "DB23_AlarmProgram".dbx1_0 )
   END_RUNG
   RUNG wire#w1
      Contact( "M16.2" )
   END_RUNG wire#w2
   RUNG wire#w1
      Contact( "M15.7" )
      I_Contact( "E22" )
   END_RUNG wire#w3
   // the same network as SCL:
   IF "M0.0" AND "DB03_Machine".dbx4_2 AND ((("M16.0" OR "M16.2") AND "DB03_Machine".dbx4_2 AND NOT "M15.7" AND NOT "E22") OR ("M15.7" AND NOT "E22")) THEN
       "DB23_AlarmProgram".dbx1_0 := TRUE;
   END_IF;
END_REGION

REGION Network 8: Alarm 10: The spool carriage encoder is not running (Technoplat)
   RUNG wire#powerrail
      Contact( "DB05_SpoolCarriagePos".dbx3_1 )
      I_Contact( "M15.1" )
      { S7_Templates := "SrcType := Int" } GE_Contact(in1 := "DB05_SpoolCarriagePos".dbw6, in2 := "DB20_DisplaySysdata".dbw8)
      S_Coil( "DB23_AlarmProgram".dbx1_1 )
   END_RUNG
   // the same network as SCL:
   IF "DB05_SpoolCarriagePos".dbx3_1 AND NOT "M15.1" AND ("DB05_SpoolCarriagePos".dbw6 >= "DB20_DisplaySysdata".dbw8) THEN
       "DB23_AlarmProgram".dbx1_1 := TRUE;
   END_IF;
END_REGION

REGION Network 9: Alarm 11: The table rotation encoder is not running (Technoplat)
   RUNG wire#powerrail
      Contact( "DB09_TablePos".dbx3_1 )
      I_Contact( "M15.7" )
      { S7_Templates := "SrcType := Int" } GE_Contact(in1 := "DB09_TablePos".dbw6, in2 := "DB20_DisplaySysdata".dbw88)
      S_Coil( "DB23_AlarmProgram".dbx1_2 )
   END_RUNG
   // the same network as SCL:
   IF "DB09_TablePos".dbx3_1 AND NOT "M15.7" AND ("DB09_TablePos".dbw6 >= "DB20_DisplaySysdata".dbw88) THEN
       "DB23_AlarmProgram".dbx1_2 := TRUE;
   END_IF;
END_REGION

REGION Network 10: Alarm 12: Overspeed for arm rotation (Technoplat)
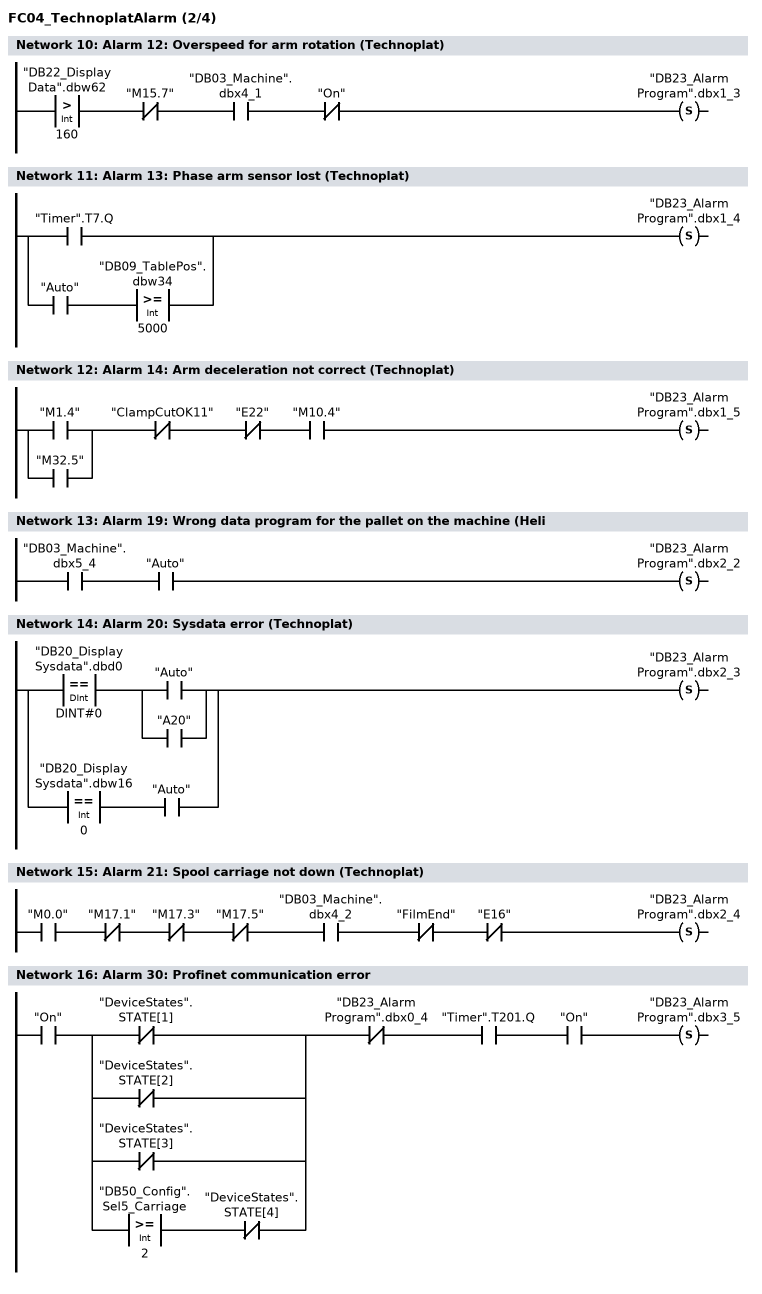
   RUNG wire#powerrail
      { S7_Templates := "SrcType := Int" } GT_Contact(in1 := "DB22_DisplayData".dbw62, in2 := 160)
      I_Contact( "M15.7" )
      Contact( "DB03_Machine".dbx4_1 )
      I_Contact( "On" )
      S_Coil( "DB23_AlarmProgram".dbx1_3 )
   END_RUNG
   // the same network as SCL:
   IF ("DB22_DisplayData".dbw62 > 160) AND NOT "M15.7" AND "DB03_Machine".dbx4_1 AND NOT "On" THEN
       "DB23_AlarmProgram".dbx1_3 := TRUE;
   END_IF;
END_REGION

REGION Network 11: Alarm 13: Phase arm sensor lost (Technoplat)
   RUNG wire#powerrail
      Contact( "Timer".T7.Q )
      wire#w1
      S_Coil( "DB23_AlarmProgram".dbx1_4 )
   END_RUNG
   RUNG wire#powerrail
      Contact( "Auto" )
      { S7_Templates := "SrcType := Int" } GE_Contact(in1 := "DB09_TablePos".dbw34, in2 := 5000)
   END_RUNG wire#w1
   // the same network as SCL:
   IF "Timer".T7.Q OR ("Auto" AND ("DB09_TablePos".dbw34 >= 5000)) THEN
       "DB23_AlarmProgram".dbx1_4 := TRUE;
   END_IF;
END_REGION

REGION Network 12: Alarm 14: Arm deceleration not correct (Technoplat)
   RUNG wire#powerrail
      Contact( "M1.4" )
      wire#w1
      I_Contact( "ClampCutOK11" )
      I_Contact( "E22" )
      Contact( "M10.4" )
      S_Coil( "DB23_AlarmProgram".dbx1_5 )
   END_RUNG
   RUNG wire#powerrail
      Contact( "M32.5" )
   END_RUNG wire#w1
   // the same network as SCL:
   IF ("M1.4" OR "M32.5") AND NOT "ClampCutOK11" AND NOT "E22" AND "M10.4" THEN
       "DB23_AlarmProgram".dbx1_5 := TRUE;
   END_IF;
END_REGION

REGION Network 13: Alarm 19: Wrong data program for the pallet on the machine (Heli
   RUNG wire#powerrail
      Contact( "DB03_Machine".dbx5_4 )
      Contact( "Auto" )
      S_Coil( "DB23_AlarmProgram".dbx2_2 )
   END_RUNG
   // the same network as SCL:
   IF "DB03_Machine".dbx5_4 AND "Auto" THEN "DB23_AlarmProgram".dbx2_2 := TRUE; END_IF;
END_REGION

REGION Network 14: Alarm 20: Sysdata error (Technoplat)
   RUNG wire#powerrail
      { S7_Templates := "SrcType := DInt" } EQ_Contact(in1 := "DB20_DisplaySysdata".dbd0, in2 := DINT#0)
      wire#w1
      Contact( "Auto" )
      wire#w2
      S_Coil( "DB23_AlarmProgram".dbx2_3 )
   END_RUNG
   RUNG wire#w1
      Contact( "A20" )
   END_RUNG wire#w2
   RUNG wire#powerrail
      { S7_Templates := "SrcType := Int" } EQ_Contact(in1 := "DB20_DisplaySysdata".dbw16, in2 := 0)
      Contact( "Auto" )
   END_RUNG wire#w2
   // the same network as SCL:
   IF (("DB20_DisplaySysdata".dbd0 = DINT#0) AND ("Auto" OR "A20")) OR (("DB20_DisplaySysdata".dbw16 = 0) AND "Auto") THEN
       "DB23_AlarmProgram".dbx2_3 := TRUE;
   END_IF;
END_REGION

REGION Network 15: Alarm 21: Spool carriage not down (Technoplat)
   RUNG wire#powerrail
      Contact( "M0.0" )
      I_Contact( "M17.1" )
      I_Contact( "M17.3" )
      I_Contact( "M17.5" )
      Contact( "DB03_Machine".dbx4_2 )
      I_Contact( "FilmEnd" )
      I_Contact( "E16" )
      S_Coil( "DB23_AlarmProgram".dbx2_4 )
   END_RUNG
   // the same network as SCL:
   IF "M0.0" AND NOT "M17.1" AND NOT "M17.3" AND NOT "M17.5" AND "DB03_Machine".dbx4_2 AND NOT "FilmEnd" AND NOT "E16" THEN
       "DB23_AlarmProgram".dbx2_4 := TRUE;
   END_IF;
END_REGION

REGION Network 16: Alarm 30: Profinet communication error
   RUNG wire#powerrail
      Contact( "On" )
      wire#w1
      I_Contact( "DeviceStates".STATE[1] )
      wire#w2
      I_Contact( "DB23_AlarmProgram".dbx0_4 )
      Contact( "Timer".T201.Q )
      Contact( "On" )
      S_Coil( "DB23_AlarmProgram".dbx3_5 )
   END_RUNG
   RUNG wire#w1
      I_Contact( "DeviceStates".STATE[2] )
   END_RUNG wire#w2
   RUNG wire#w1
      I_Contact( "DeviceStates".STATE[3] )
   END_RUNG wire#w2
   RUNG wire#w1
      { S7_Templates := "SrcType := Int" } GE_Contact(in1 := "DB50_Config".Sel5_Carriage, in2 := 2)
      I_Contact( "DeviceStates".STATE[4] )
   END_RUNG wire#w2
   // the same network as SCL:
   IF "On" AND (NOT "DeviceStates".STATE[1] OR NOT "DeviceStates".STATE[2] OR NOT "DeviceStates".STATE[3] OR (("DB50_Config".Sel5_Carriage >= 2) AND NOT "DeviceStates".STATE[4])) AND NOT "DB23_AlarmProgram".dbx0_4 AND "Timer".T201.Q AND "On" THEN
       "DB23_AlarmProgram".dbx3_5 := TRUE;
   END_IF;
END_REGION

REGION Network 17: Alarm 31: Modbus communication error
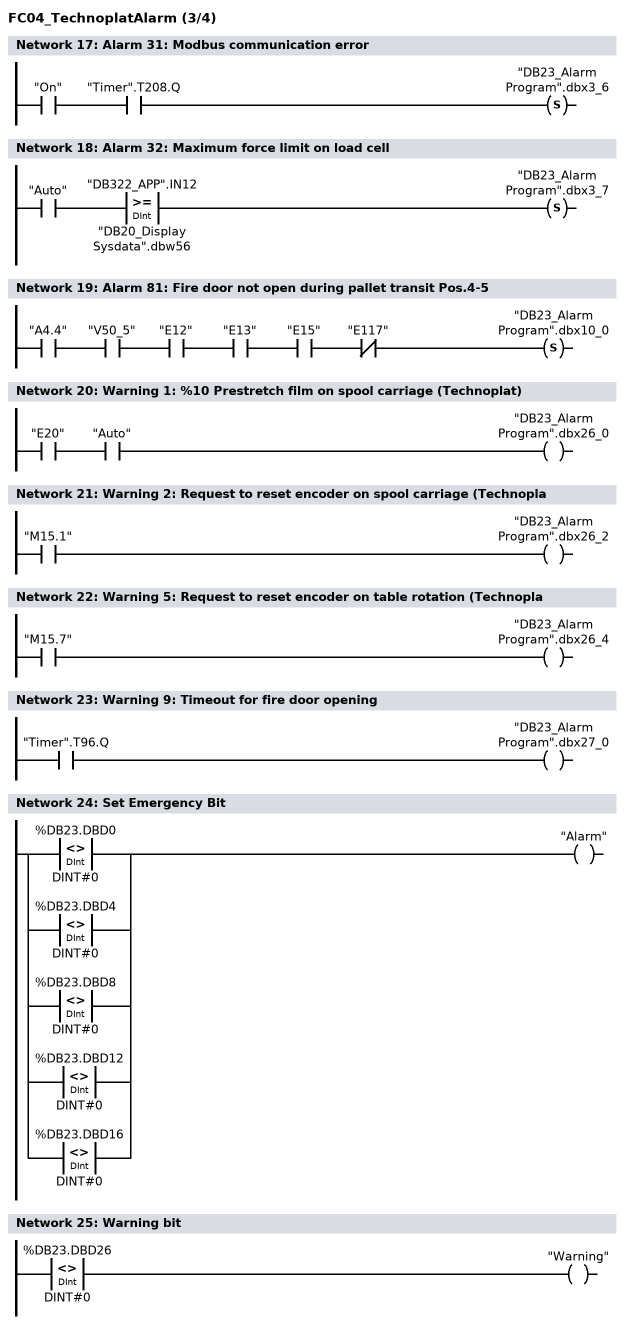
   RUNG wire#powerrail
      Contact( "On" )
      Contact( "Timer".T208.Q )
      S_Coil( "DB23_AlarmProgram".dbx3_6 )
   END_RUNG
   // the same network as SCL:
   IF "On" AND "Timer".T208.Q THEN "DB23_AlarmProgram".dbx3_6 := TRUE; END_IF;
END_REGION

REGION Network 18: Alarm 32: Maximum force limit on load cell
   RUNG wire#powerrail
      Contact( "Auto" )
      { S7_Templates := "SrcType := DInt" } GE_Contact(in1 := "DB322_APP".IN12, in2 := "DB20_DisplaySysdata".dbw56)
      S_Coil( "DB23_AlarmProgram".dbx3_7 )
   END_RUNG
   // the same network as SCL:
   IF "Auto" AND ("DB322_APP".IN12 >= "DB20_DisplaySysdata".dbw56) THEN
       "DB23_AlarmProgram".dbx3_7 := TRUE;
   END_IF;
END_REGION

REGION Network 19: Alarm 81: Fire door not open during pallet transit Pos.4-5
   RUNG wire#powerrail
      Contact( "A4.4" )
      Contact( "V50_5" )
      Contact( "E12" )
      Contact( "E13" )
      Contact( "E15" )
      I_Contact( "E117" )
      S_Coil( "DB23_AlarmProgram".dbx10_0 )
   END_RUNG
   // the same network as SCL:
   IF "A4.4" AND "V50_5" AND "E12" AND "E13" AND "E15" AND NOT "E117" THEN
       "DB23_AlarmProgram".dbx10_0 := TRUE;
   END_IF;
END_REGION

REGION Network 20: Warning 1: %10 Prestretch film on spool carriage (Technoplat)
   RUNG wire#powerrail
      Contact( "E20" )
      Contact( "Auto" )
      Coil( "DB23_AlarmProgram".dbx26_0 )
   END_RUNG
   // the same network as SCL:
   "DB23_AlarmProgram".dbx26_0 := "E20" AND "Auto";
END_REGION

REGION Network 21: Warning 2: Request to reset encoder on spool carriage (Technopla
   RUNG wire#powerrail
      Contact( "M15.1" )
      Coil( "DB23_AlarmProgram".dbx26_2 )
   END_RUNG
   // the same network as SCL:
   "DB23_AlarmProgram".dbx26_2 := "M15.1";
END_REGION

REGION Network 22: Warning 5: Request to reset encoder on table rotation (Technopla
   RUNG wire#powerrail
      Contact( "M15.7" )
      Coil( "DB23_AlarmProgram".dbx26_4 )
   END_RUNG
   // the same network as SCL:
   "DB23_AlarmProgram".dbx26_4 := "M15.7";
END_REGION

REGION Network 23: Warning 9: Timeout for fire door opening
   RUNG wire#powerrail
      Contact( "Timer".T96.Q )
      Coil( "DB23_AlarmProgram".dbx27_0 )
   END_RUNG
   // the same network as SCL:
   "DB23_AlarmProgram".dbx27_0 := "Timer".T96.Q;
END_REGION

REGION Network 24: Set Emergency Bit
   RUNG wire#powerrail
      { S7_Templates := "SrcType := DInt" } NE_Contact(in1 := %DB23.DBD0, in2 := DINT#0)
      wire#w1
      Coil( "Alarm" )
   END_RUNG
   RUNG wire#powerrail
      { S7_Templates := "SrcType := DInt" } NE_Contact(in1 := %DB23.DBD4, in2 := DINT#0)
   END_RUNG wire#w1
   RUNG wire#powerrail
      { S7_Templates := "SrcType := DInt" } NE_Contact(in1 := %DB23.DBD8, in2 := DINT#0)
   END_RUNG wire#w1
   RUNG wire#powerrail
      { S7_Templates := "SrcType := DInt" } NE_Contact(in1 := %DB23.DBD12, in2 := DINT#0)
   END_RUNG wire#w1
   RUNG wire#powerrail
      { S7_Templates := "SrcType := DInt" } NE_Contact(in1 := %DB23.DBD16, in2 := DINT#0)
   END_RUNG wire#w1
   // the same network as SCL:
   "Alarm" := (%DB23.DBD0 <> DINT#0) OR (%DB23.DBD4 <> DINT#0) OR (%DB23.DBD8 <> DINT#0) OR (%DB23.DBD12 <> DINT#0) OR (%DB23.DBD16 <> DINT#0);
END_REGION

REGION Network 25: Warning bit
   RUNG wire#powerrail
      { S7_Templates := "SrcType := DInt" } NE_Contact(in1 := %DB23.DBD26, in2 := DINT#0)
      Coil( "Warning" )
   END_RUNG
   // the same network as SCL:
   "Warning" := %DB23.DBD26 <> DINT#0;
END_REGION

REGION Network 26: First cycle
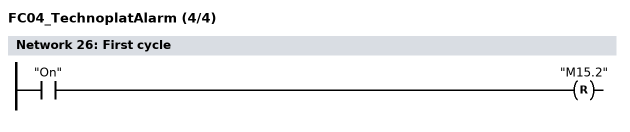
   RUNG wire#powerrail
      Contact( "On" )
      R_Coil( "M15.2" )
   END_RUNG
   // the same network as SCL:
   IF "On" THEN "M15.2" := FALSE; END_IF;
END_REGION
END_FUNCTION

ORGANIZATION_BLOCK "Cyclic interrupt"   // OB30, LAD, CyclicInterrupt
TITLE = Rampa tiro
{ S7_Optimized_Access := 'TRUE' }
VERSION : 0.1
// Rampa per raggiungere tiro obiettivo e zero (0-20@100ms;20-100@20ms->3600ms)
// stored: AutoNumber true, IsIECCheckEnabled false, SetENOAutomatically false
   VAR_INPUT
      Initial_Call : Bool;   // Initial call of this OB
      Event_Count : Int;   // Events discarded
   END_VAR
   VAR_TEMP
      TempDint : DInt;
      TempDint_2 : DInt;
      TempInt : Int;
   END_VAR
   VAR_TEMP   // added for the SCL form of the ladder/FBD networks
      _w1 : Bool;
      _w2 : Bool;
   END_VAR
BEGIN

REGION Network 1: Impulso ogni 20ms (OB30)
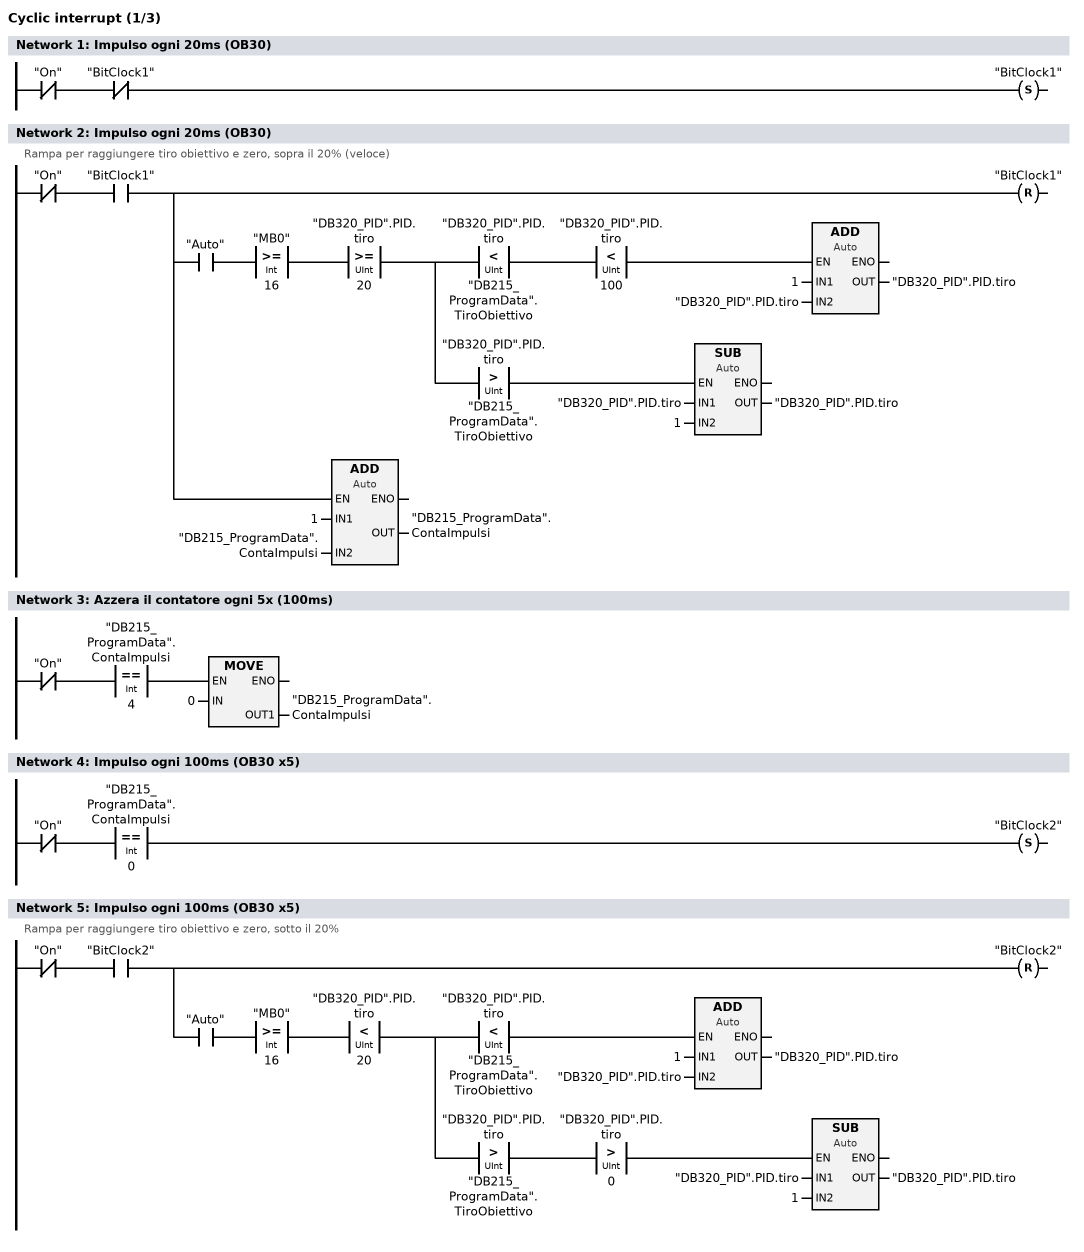
   RUNG wire#powerrail
      I_Contact( "On" )
      I_Contact( "BitClock1" )
      S_Coil( "BitClock1" )
   END_RUNG
   // the same network as SCL:
   IF NOT "On" AND NOT "BitClock1" THEN "BitClock1" := TRUE; END_IF;
END_REGION

REGION Network 2: Impulso ogni 20ms (OB30)
   // Rampa per raggiungere tiro obiettivo e zero, sopra il 20% (veloce)
   RUNG wire#powerrail
      I_Contact( "On" )
      Contact( "BitClock1" )
      wire#w1
      R_Coil( "BitClock1" )
   END_RUNG
   RUNG wire#w1
      Contact( "Auto" )
      { S7_Templates := "SrcType := Int" } GE_Contact(in1 := "MB0", in2 := 16)
      { S7_Templates := "SrcType := UInt" } GE_Contact(in1 := "DB320_PID".PID.tiro, in2 := 20)
      wire#w2
      { S7_Templates := "SrcType := UInt" } LT_Contact(in1 := "DB320_PID".PID.tiro, in2 := "DB215_ProgramData".TiroObiettivo)
      { S7_Templates := "SrcType := UInt" } LT_Contact(in1 := "DB320_PID".PID.tiro, in2 := 100)
      Add(in1 := 1, in2 := "DB320_PID".PID.tiro, out => "DB320_PID".PID.tiro)
   END_RUNG
   RUNG wire#w2
      { S7_Templates := "SrcType := UInt" } GT_Contact(in1 := "DB320_PID".PID.tiro, in2 := "DB215_ProgramData".TiroObiettivo)
      Sub(in1 := "DB320_PID".PID.tiro, in2 := 1, out => "DB320_PID".PID.tiro)
   END_RUNG
   RUNG wire#w1
      Add(in1 := 1, in2 := "DB215_ProgramData".ContaImpulsi, out => "DB215_ProgramData".ContaImpulsi)
   END_RUNG
   // the same network as SCL:
   #_w1 := NOT "On" AND "BitClock1";
   IF #_w1 THEN "BitClock1" := FALSE; END_IF;
   #_w2 := #_w1 AND "Auto" AND ("MB0" >= 16) AND ("DB320_PID".PID.tiro >= 20);
   IF #_w2 AND ("DB320_PID".PID.tiro < "DB215_ProgramData".TiroObiettivo) AND ("DB320_PID".PID.tiro < 100) THEN
       "DB320_PID".PID.tiro := 1 + "DB320_PID".PID.tiro;
   END_IF;
   IF #_w2 AND ("DB320_PID".PID.tiro > "DB215_ProgramData".TiroObiettivo) THEN
       "DB320_PID".PID.tiro := "DB320_PID".PID.tiro - 1;
   END_IF;
   IF #_w1 THEN "DB215_ProgramData".ContaImpulsi := 1 + "DB215_ProgramData".ContaImpulsi; END_IF;
END_REGION

REGION Network 3: Azzera il contatore ogni 5x (100ms)
   RUNG wire#powerrail
      I_Contact( "On" )
      { S7_Templates := "SrcType := Int" } EQ_Contact(in1 := "DB215_ProgramData".ContaImpulsi, in2 := 4)
      Move(in := 0, out1 => "DB215_ProgramData".ContaImpulsi)
   END_RUNG
   // the same network as SCL:
   IF NOT "On" AND ("DB215_ProgramData".ContaImpulsi = 4) THEN "DB215_ProgramData".ContaImpulsi := 0; END_IF;
END_REGION

REGION Network 4: Impulso ogni 100ms (OB30 x5)
   RUNG wire#powerrail
      I_Contact( "On" )
      { S7_Templates := "SrcType := Int" } EQ_Contact(in1 := "DB215_ProgramData".ContaImpulsi, in2 := 0)
      S_Coil( "BitClock2" )
   END_RUNG
   // the same network as SCL:
   IF NOT "On" AND ("DB215_ProgramData".ContaImpulsi = 0) THEN "BitClock2" := TRUE; END_IF;
END_REGION

REGION Network 5: Impulso ogni 100ms (OB30 x5)
   // Rampa per raggiungere tiro obiettivo e zero, sotto il 20%
   RUNG wire#powerrail
      I_Contact( "On" )
      Contact( "BitClock2" )
      wire#w1
      R_Coil( "BitClock2" )
   END_RUNG
   RUNG wire#w1
      Contact( "Auto" )
      { S7_Templates := "SrcType := Int" } GE_Contact(in1 := "MB0", in2 := 16)
      { S7_Templates := "SrcType := UInt" } LT_Contact(in1 := "DB320_PID".PID.tiro, in2 := 20)
      wire#w2
      { S7_Templates := "SrcType := UInt" } LT_Contact(in1 := "DB320_PID".PID.tiro, in2 := "DB215_ProgramData".TiroObiettivo)
      Add(in1 := 1, in2 := "DB320_PID".PID.tiro, out => "DB320_PID".PID.tiro)
   END_RUNG
   RUNG wire#w2
      { S7_Templates := "SrcType := UInt" } GT_Contact(in1 := "DB320_PID".PID.tiro, in2 := "DB215_ProgramData".TiroObiettivo)
      { S7_Templates := "SrcType := UInt" } GT_Contact(in1 := "DB320_PID".PID.tiro, in2 := 0)
      Sub(in1 := "DB320_PID".PID.tiro, in2 := 1, out => "DB320_PID".PID.tiro)
   END_RUNG
   // the same network as SCL:
   #_w1 := NOT "On" AND "BitClock2";
   IF #_w1 THEN "BitClock2" := FALSE; END_IF;
   #_w2 := #_w1 AND "Auto" AND ("MB0" >= 16) AND ("DB320_PID".PID.tiro < 20);
   IF #_w2 AND ("DB320_PID".PID.tiro < "DB215_ProgramData".TiroObiettivo) THEN
       "DB320_PID".PID.tiro := 1 + "DB320_PID".PID.tiro;
   END_IF;
   IF #_w2 AND ("DB320_PID".PID.tiro > "DB215_ProgramData".TiroObiettivo) AND ("DB320_PID".PID.tiro > 0) THEN
       "DB320_PID".PID.tiro := "DB320_PID".PID.tiro - 1;
   END_IF;
END_REGION

REGION Network 7: Arm rotation and top carriage speed change for DAC M20
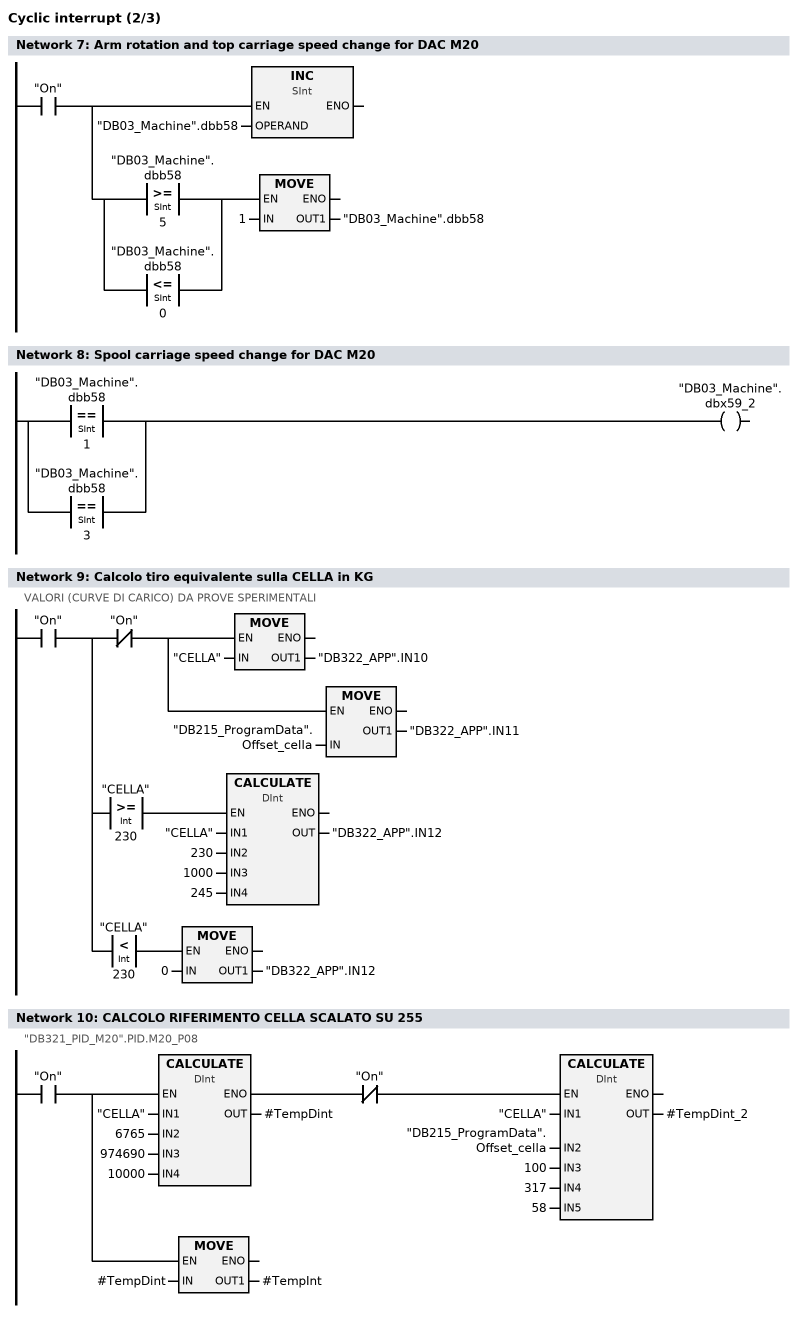
   RUNG wire#powerrail
      Contact( "On" )
      wire#w1
      { S7_Templates := "DestType := SInt"; S7_GenerateENO := "TRUE" } Inc( "DB03_Machine".dbb58 )
   END_RUNG
   RUNG wire#w1
      { S7_Templates := "SrcType := SInt" } GE_Contact(in1 := "DB03_Machine".dbb58, in2 := 5)
      wire#w2
      { S7_GenerateENO := "TRUE" } Move(in := 1, out1 => "DB03_Machine".dbb58)
   END_RUNG
   RUNG wire#w1
      { S7_Templates := "SrcType := SInt" } LE_Contact(in1 := "DB03_Machine".dbb58, in2 := 0)
   END_RUNG wire#w2
   // the same network as SCL:
   IF "On" THEN "DB03_Machine".dbb58 := "DB03_Machine".dbb58 + 1; END_IF;
   IF "On" AND (("DB03_Machine".dbb58 >= 5) OR ("DB03_Machine".dbb58 <= 0)) THEN
       "DB03_Machine".dbb58 := 1;
   END_IF;
END_REGION

REGION Network 8: Spool carriage speed change for DAC M20
   RUNG wire#powerrail
      { S7_Templates := "SrcType := SInt" } EQ_Contact(in1 := "DB03_Machine".dbb58, in2 := 1)
      wire#w1
      Coil( "DB03_Machine".dbx59_2 )
   END_RUNG
   RUNG wire#powerrail
      { S7_Templates := "SrcType := SInt" } EQ_Contact(in1 := "DB03_Machine".dbb58, in2 := 3)
   END_RUNG wire#w1
   // the same network as SCL:
   "DB03_Machine".dbx59_2 := ("DB03_Machine".dbb58 = 1) OR ("DB03_Machine".dbb58 = 3);
END_REGION

REGION Network 9: Calcolo tiro equivalente sulla CELLA in KG
   // VALORI (CURVE DI CARICO) DA PROVE SPERIMENTALI
   RUNG wire#powerrail
      Contact( "On" )
      wire#w1
      I_Contact( "On" )
      wire#w2
      Move(in := "CELLA", out1 => "DB322_APP".IN10)
   END_RUNG
   RUNG wire#w2
      Move(in := "DB215_ProgramData".Offset_cella, out1 => "DB322_APP".IN11)
   END_RUNG
   RUNG wire#w1
      { S7_Templates := "SrcType := Int" } GE_Contact(in1 := "CELLA", in2 := 230)
      { S7_Templates := "SrcType := DInt"; S7_Expression := "((IN1-IN2)*IN3)/IN4" } Calculate(in1 := "CELLA", in2 := 230, in3 := 1000, in4 := 245, out => "DB322_APP".IN12)
   END_RUNG
   RUNG wire#w1
      { S7_Templates := "SrcType := Int" } LT_Contact(in1 := "CELLA", in2 := 230)
      Move(in := 0, out1 => "DB322_APP".IN12)
   END_RUNG
   // the same network as SCL:
   IF "On" AND NOT "On" THEN
       "DB322_APP".IN10 := "CELLA";
       "DB322_APP".IN11 := "DB215_ProgramData".Offset_cella;
   END_IF;
   IF "On" AND ("CELLA" >= 230) THEN "DB322_APP".IN12 := (("CELLA"-230)*1000)/245; END_IF;
   IF "On" AND ("CELLA" < 230) THEN "DB322_APP".IN12 := 0; END_IF;
END_REGION

REGION Network 10: CALCOLO RIFERIMENTO CELLA SCALATO SU 255
   // "DB321_PID_M20".PID.M20_P08
   RUNG wire#powerrail
      Contact( "On" )
      wire#w1
      { S7_Templates := "SrcType := DInt"; S7_Expression := "(IN1*IN2-IN3)/IN4" } Calculate(in1 := "CELLA", in2 := 6765, in3 := 974690, in4 := 10000, out => #TempDint)
      I_Contact( "On" )
      { S7_Templates := "SrcType := DInt"; S7_Expression := "((IN1-IN2)*IN3/IN4)+IN5" } Calculate(in1 := "CELLA", in2 := "DB215_ProgramData".Offset_cella, in3 := 100, in4 := 317, in5 := 58, out => #TempDint_2)
   END_RUNG
   RUNG wire#w1
      Move(in := #TempDint, out1 => #TempInt)
   END_RUNG
   // the same network as SCL:
   IF "On" THEN #TempDint := ("CELLA"*6765-974690)/10000; END_IF;
   IF "On" AND NOT "On" THEN #TempDint_2 := (("CELLA"-"DB215_ProgramData".Offset_cella)*100/317)+58; END_IF;
   IF "On" THEN #TempInt := #TempDint; END_IF;
END_REGION

REGION Network 11: M20
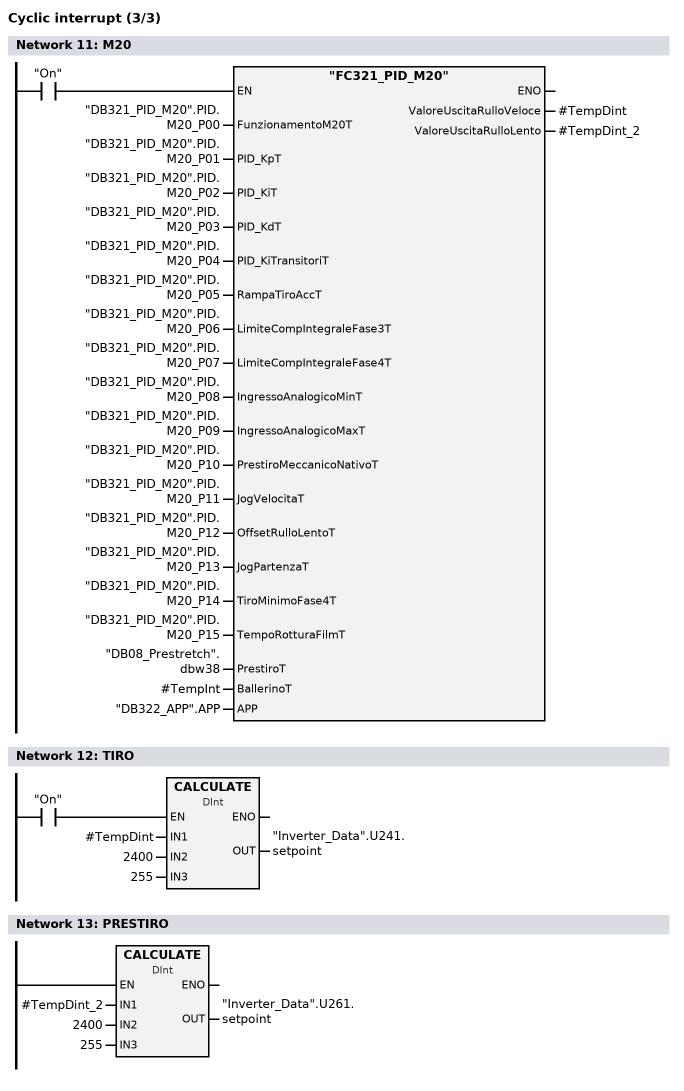
   RUNG wire#powerrail
      Contact( "On" )
      "FC321_PID_M20"(FunzionamentoM20T := "DB321_PID_M20".PID.M20_P00, PID_KpT := "DB321_PID_M20".PID.M20_P01, PID_KiT := "DB321_PID_M20".PID.M20_P02, PID_KdT := "DB321_PID_M20".PID.M20_P03, PID_KiTransitoriT := "DB321_PID_M20".PID.M20_P04, RampaTiroAccT := "DB321_PID_M20".PID.M20_P05, LimiteCompIntegraleFase3T := "DB321_PID_M20".PID.M20_P06, LimiteCompIntegraleFase4T := "DB321_PID_M20".PID.M20_P07, IngressoAnalogicoMinT := "DB321_PID_M20".PID.M20_P08, IngressoAnalogicoMaxT := "DB321_PID_M20".PID.M20_P09, PrestiroMeccanicoNativoT := "DB321_PID_M20".PID.M20_P10, JogVelocitaT := "DB321_PID_M20".PID.M20_P11, OffsetRulloLentoT := "DB321_PID_M20".PID.M20_P12, JogPartenzaT := "DB321_PID_M20".PID.M20_P13, TiroMinimoFase4T := "DB321_PID_M20".PID.M20_P14, TempoRotturaFilmT := "DB321_PID_M20".PID.M20_P15, PrestiroT := "DB08_Prestretch".dbw38, BallerinoT := #TempInt, APP := "DB322_APP".APP, ValoreUscitaRulloVeloce => #TempDint, ValoreUscitaRulloLento => #TempDint_2)
   END_RUNG
   // the same network as SCL:
   IF "On" THEN
       "FC321_PID_M20"(FunzionamentoM20T := "DB321_PID_M20".PID.M20_P00,
                       PID_KpT := "DB321_PID_M20".PID.M20_P01,
                       PID_KiT := "DB321_PID_M20".PID.M20_P02,
                       PID_KdT := "DB321_PID_M20".PID.M20_P03,
                       PID_KiTransitoriT := "DB321_PID_M20".PID.M20_P04,
                       RampaTiroAccT := "DB321_PID_M20".PID.M20_P05,
                       LimiteCompIntegraleFase3T := "DB321_PID_M20".PID.M20_P06,
                       LimiteCompIntegraleFase4T := "DB321_PID_M20".PID.M20_P07,
                       IngressoAnalogicoMinT := "DB321_PID_M20".PID.M20_P08,
                       IngressoAnalogicoMaxT := "DB321_PID_M20".PID.M20_P09,
                       PrestiroMeccanicoNativoT := "DB321_PID_M20".PID.M20_P10,
                       JogVelocitaT := "DB321_PID_M20".PID.M20_P11,
                       OffsetRulloLentoT := "DB321_PID_M20".PID.M20_P12,
                       JogPartenzaT := "DB321_PID_M20".PID.M20_P13,
                       TiroMinimoFase4T := "DB321_PID_M20".PID.M20_P14,
                       TempoRotturaFilmT := "DB321_PID_M20".PID.M20_P15,
                       PrestiroT := "DB08_Prestretch".dbw38,
                       BallerinoT := #TempInt,
                       APP := "DB322_APP".APP,
                       ValoreUscitaRulloVeloce => #TempDint,
                       ValoreUscitaRulloLento => #TempDint_2);
   END_IF;
END_REGION

REGION Network 12: TIRO
   RUNG wire#powerrail
      Contact( "On" )
      { S7_Templates := "SrcType := DInt"; S7_Expression := "IN1*IN2/IN3" } Calculate(in1 := #TempDint, in2 := 2400, in3 := 255, out => "Inverter_Data".U241.setpoint)
   END_RUNG
   // the same network as SCL:
   IF "On" THEN "Inverter_Data".U241.setpoint := #TempDint*2400/255; END_IF;
END_REGION

REGION Network 13: PRESTIRO
   RUNG wire#powerrail
      { S7_Templates := "SrcType := DInt"; S7_Expression := "IN1*IN2/IN3" } Calculate(in1 := #TempDint_2, in2 := 2400, in3 := 255, out => "Inverter_Data".U261.setpoint)
   END_RUNG
   // the same network as SCL:
   "Inverter_Data".U261.setpoint := #TempDint_2*2400/255;
END_REGION
END_ORGANIZATION_BLOCK

FUNCTION "FC321_PID_M20" : Void
{ S7_Optimized_Access := 'TRUE' }
VERSION : 0.1
   VAR_INPUT 
      FunzionamentoM20T : Int;
      PID_KpT : Int;
      PID_KiT : Int;
      PID_KdT : Int;
      PID_KiTransitoriT : Int;
      RampaTiroAccT : Int;
      LimiteCompIntegraleFase3T : Int;
      LimiteCompIntegraleFase4T : Int;
      IngressoAnalogicoMinT : Int;
      IngressoAnalogicoMaxT : Int;
      PrestiroMeccanicoNativoT : Int;
      JogVelocitaT : Int;
      OffsetRulloLentoT : Int;
      JogPartenzaT : Int;
      TiroMinimoFase4T : Int;
      TempoRotturaFilmT : Int;
      PrestiroT : Int;
      BallerinoT : Int;
   END_VAR

   VAR_OUTPUT 
      ValoreUscitaRulloVeloce : DInt;
      ValoreUscitaRulloLento : DInt;
   END_VAR

   VAR_IN_OUT 
      APP : "APP";
   END_VAR

   VAR_TEMP 
      PID_ComponenteProporzionale : DInt;
      PID_ComponenteIntegrale : DInt;
      PID_ComponenteDerivativa : DInt;
      Tiro : Int;
      Tiro1 : Int;
      Tiro2 : Int;
      TiroPrecedente : Int;
      TiroAppoggio : Int;
      ErroreAttuale : Int;
      ErrorePrecedente : Int;
      PID_Kp : Int;
      PID_Ki : Int;
      PID_Kd : Int;
      SetpointTiro : Int;
      SetpointTiroRampa : Int;
      TransitorioInizialeFase1 : Int;
      TransitorioFase3 : Int;
      TransitorioFase4 : Int;
      VelocitaRotazione : Int;
      VelocitaRotazioneFase2 : Int;
      VelocitaRotazioneAppoggio1 : Int;
      VelocitaRotazioneAppoggio2 : Int;
      Fase1OneShoot : Int;
      Fase2OneShoot : Int;
      Fase3OneShoot : Int;
      Fase4OneShoot : Int;
      ArrestoRepentinoOneShoot : Int;
      TiroFase1 : Int;
      TempIntero : Int;
      Fase : Int;
      BallerinoPrecedente : Array[0..2] of Int;
      LimiteComponenteIntegrale : Int;
      TiroRichiesto : Int;
      TimerArrestoRepentino : Int;
      TiroMinimoArrestoRepentino : Int;
      VariazioneTiro : Int;
      TimerFase2 : Int;
      TempoRotturaFilm : Int;
      TimerFase4 : Int;
      TiroMinimoFase4 : Int;
      PID_Uscita : DInt;
      PrestiroRichiesto : DInt;
      PrestiroAppoggio : Real;
   END_VAR

   VAR CONSTANT 
      PID_LimiteSuperioreIntegrale : DInt := 23000;
      PID_LimiteInferioreIntegrale : DInt := 0;
      PID_LimiteSuperioreDerivativa : DInt := 6000;
      PID_LimiteInferioreDerivativa : DInt := -6000;
      PID_LimiteSuperioreUscita : DInt := 255;
      PID_LimiteInferioreUscita : DInt := 0;
   END_VAR


BEGIN
	// Devono esserci due letture uguali per cambiare il valore di tiro. Serve a filtrare letture spurie
	//
	#APP.Tiro1 := "DB08_Prestretch".dbw18; //val_parametro[22];
	//
	IF (#APP.Tiro1 = #APP.Tiro2) THEN
	    #APP.Tiro := #APP.#Tiro1;
	END_IF;
	//
	#APP.Tiro2 := #APP.#Tiro1;
	//
	#APP.VelocitaRotazione := "DB09_TablePos".dbw10; //val_parametro[20];
	//
	// Fase 1:  Accelerazione
	//***********************
	IF (#APP.Tiro = 206) THEN
	    #APP.Fase := 1;
	    //Inizializzazione Fase 1
	    IF (#APP.Fase1OneShoot = 0) THEN
	        #APP.SetpointTiroRampa := #BallerinoT * 10;
	        #APP.TransitorioInizialeFase1 := 1;
	        #APP.Fase1OneShoot := 1;
	        #APP.PID_ComponenteIntegrale := #APP.PID_ComponenteIntegrale + #JogPartenzaT * 100; //Incremento di componente integrale per limitare tiri alti alla partenza 
	    END_IF;
	    //
	    #APP.VariazioneTiro := #BallerinoT-#APP.BallerinoPrecedente[2];
	    //#APP.VariazioneTiro := (#BallerinoT - #APP.BallPrec_2);
	    #APP.PID_Kp := #PID_KpT*2;
	    #APP.PID_Ki := #PID_KiT*2;
	    #APP.PID_Kd := #PID_KdT*3;
	    //
	    IF (#APP.VariazioneTiro < 0) THEN
	        #APP.PID_Kd := 0;
	    END_IF;
	    //
	    IF (#APP.TiroFase1 = 0) THEN
	        #APP.TiroFase1 := 5;
	    END_IF;
	    //
	    #APP.SetpointTiro := ((#IngressoAnalogicoMaxT-#IngressoAnalogicoMinT)*#APP.TiroFase1/100)+#IngressoAnalogicoMinT;
	    //
	    //Incremento componente integrale durante la fase di accelerazione per ridurre l'errore sul tiro desiderato
	    IF (#APP.VariazioneTiro > 0 AND #APP.ErroreAttuale > 0) THEN
	        IF (#FunzionamentoM20T = 0) THEN
	            #APP.PID_ComponenteIntegrale := #APP.PID_ComponenteIntegrale + #PID_KpT * #APP.ErroreAttuale / 4;
	        ELSE //(#APP.FunzionamentoM20T == 1)
	            #APP.PID_ComponenteIntegrale := #APP.PID_ComponenteIntegrale + #PID_KpT * #APP.ErroreAttuale / 10;
	        END_IF;
	    END_IF;
	    //Rampa di tiro per tiri alti
	    IF (#APP.TransitorioInizialeFase1 = 1) THEN
	        IF (#APP.SetpointTiroRampa / 10 < #APP.SetpointTiro) THEN
	            #APP.SetpointTiroRampa := #APP.SetpointTiroRampa + #RampaTiroAccT;
	            #APP.SetpointTiro := #APP.SetpointTiroRampa / 10;
	        ELSE
	            #APP.TransitorioInizialeFase1 := 0;
	        END_IF;
	    END_IF;
	    #APP.TiroRichiesto := #APP.TiroFase1;
	END_IF;
	//
	// Fase 2: Fasciatura a regime
	//****************************
	IF (#APP.Tiro > 0 AND #APP.Tiro <= 100) THEN
	    #APP.Fase := 2;
	    #APP.Fase4OneShoot := 0;
	    // Inizializzazione Fase 2      
	    IF (#APP.Fase2OneShoot = 0) THEN
	        #APP.VelocitaRotazioneFase2 := 0;
	        #APP.Fase2OneShoot := 1;
	// PID_ComponenteIntegrale = PID_ComponenteIntegrale+2000; //Fornisco un piccolo delta di velocita'alla partenza per evitare di tirare strattoni sul ballerino all'avvio 
	    END_IF;
	    #APP.PID_Kp := #PID_KpT;
	    #APP.PID_Ki := #PID_KiT;
	    #APP.PID_Kd := #PID_KdT;
	    IF (#APP.Tiro >= 50) THEN
	        #APP.PID_Ki := (15+20*#PID_KiT)/30; //Per tiri alti diminuisco il guadagno integrale per rendere il regolatore meno pronto e farlo oscillare meno.
	    END_IF;
	    #APP.SetpointTiro := ((#IngressoAnalogicoMaxT-#IngressoAnalogicoMinT)*#APP.Tiro/100)+#IngressoAnalogicoMinT;
	    #APP.TiroFase1 := #APP.Tiro;
	    //
	    //Velocita' di rotazione braccio nella Fase 2. Filtro di 3 scansioni
	    IF (#APP.VelocitaRotazione = #APP.VelocitaRotazioneAppoggio1 AND #APP.VelocitaRotazioneAppoggio1 = #APP.VelocitaRotazioneAppoggio2) THEN
	        #APP.VelocitaRotazioneFase2 := #APP.VelocitaRotazione;
	    END_IF;
	    #APP.VelocitaRotazioneAppoggio2 := #APP.VelocitaRotazioneAppoggio1;
	    #APP.VelocitaRotazioneAppoggio1 := #APP.VelocitaRotazione;
	    //
	    //Rottura film
	    IF (#BallerinoT < #IngressoAnalogicoMinT) THEN
	        #APP.TimerFase2 := #APP.TimerFase2 + 1;
	    ELSE
	        #APP.TimerFase2 := 0;
	    END_IF;
	    //
	    #APP.TempoRotturaFilm := #TempoRotturaFilmT*10/3; //Tempo rottura film in numero di scansioni
	    IF (#APP.TimerFase2 >= #APP.TempoRotturaFilm) THEN
	        #APP.PID_ComponenteIntegrale := 0;
	        #APP.TimerFase2 := 0;
	    END_IF;
	    #APP.TiroRichiesto := #APP.Tiro;
	END_IF;
	//
	// Fase 3: Transitorio velocita' alta -> media
	//********************************************
	IF (#APP.Tiro > 100 AND #APP.Tiro <= 200) THEN
	    #APP.Fase := 3 ;
	    #APP.Fase4OneShoot := 0;
	    //
	    // Inizializzazione Fase 3
	    IF (#APP.Fase3OneShoot = 0) THEN
	        #APP.TransitorioFase3 := 0;
	        #APP.Fase3OneShoot := 1;
	    END_IF;
	    //
	    #APP.LimiteComponenteIntegrale := #LimiteCompIntegraleFase3T*100;
	    #APP.PID_Kp := #PID_KpT;
	    #APP.PID_Ki := #PID_KiTransitoriT;
	    #APP.PID_Kd := #PID_KdT;
	    #APP.SetpointTiro := ((#IngressoAnalogicoMaxT-#IngressoAnalogicoMinT)*(#APP.Tiro-100)/100)+#IngressoAnalogicoMinT;
	    //
	    #APP.TempIntero := #APP.VelocitaRotazioneFase2*9/10;
	    IF (#APP.VelocitaRotazione < #APP.TempIntero AND #APP.TransitorioFase3 = 0) THEN
	        #APP.TransitorioFase3 := 1;
	        IF (#APP.PID_ComponenteIntegrale > #APP.LimiteComponenteIntegrale) THEN
	            #APP.PID_ComponenteIntegrale := #APP.LimiteComponenteIntegrale;
	        END_IF;
	    END_IF;
	    #APP.TiroRichiesto := #APP.Tiro-100;
	END_IF;
	//
	// Fase 4: Transitorio velocita' media -> bassa
	// ********************************************
	IF (#APP.Tiro = 201) THEN
	    #APP.Fase := 4 ;
	    // Inizializzazione Fase 4
	    IF (#APP.Fase4OneShoot = 0) THEN
	        #APP.TransitorioFase4 := 0;
	        #APP.Fase4OneShoot := 1;
	    END_IF;
	    //
	    IF (#APP.TiroPrecedente <= 100) THEN
	        #APP.TiroAppoggio := #APP.TiroPrecedente;
	    END_IF;
	    //
	    IF (#APP.TiroPrecedente > 100 AND #APP.TiroPrecedente <= 200) THEN
	        #APP.TiroAppoggio := #APP.TiroPrecedente - 100;
	    END_IF;
	    //
	    //Alzo il tiro richiesto nei primi decimi, in maniera da abbattere la componente integrale
	    #APP.TiroMinimoFase4 := #TiroMinimoFase4T;
	    //
	    IF (#APP.TiroAppoggio < #APP.TiroMinimoFase4) THEN
	        #APP.TiroAppoggio := #APP.TiroMinimoFase4;
	    END_IF;
	    //
	    #APP.SetpointTiro := ((#IngressoAnalogicoMaxT-#IngressoAnalogicoMinT)*#APP.TiroAppoggio/100)+#IngressoAnalogicoMinT;
	    //
	    #APP.LimiteComponenteIntegrale := #LimiteCompIntegraleFase4T*100;
	    #APP.PID_Kp := #PID_KpT;
	    #APP.PID_Ki := #PID_KiTransitoriT*15/10;
	    #APP.PID_Kd := #PID_KdT;
	    IF (#APP.PID_ComponenteIntegrale > #APP.LimiteComponenteIntegrale) THEN
	        #APP.PID_ComponenteIntegrale := #APP.LimiteComponenteIntegrale;
	    END_IF;
	    //
	    #APP.TransitorioFase4 := 1 ;
	    #APP.TiroRichiesto := #APP.TiroAppoggio;
	END_IF;
	//
	// Fase 0: Azzeramento del regolatore
	// **********************************
	IF (#APP.Tiro = 0) THEN
	    #APP.Fase := 0;
	    #APP.PID_ComponenteIntegrale := 0;
	    #APP.Fase1OneShoot := 0;
	    #APP.Fase2OneShoot := 0;
	    #APP.Fase3OneShoot := 0;
	    #APP.Fase4OneShoot := 0;
	    #APP.ArrestoRepentinoOneShoot := 0;
	    #APP.SetpointTiro := #BallerinoT;
	    #APP.TiroPrecedente := 0;
	    #APP.TiroFase1 := 0;
	    #APP.TiroAppoggio := 0;
	END_IF;
	//   
	// Jog in manuale
	// **************
	IF (#APP.Tiro = 210) THEN
	    #APP.PID_Kp := 0;
	    #APP.PID_Ki := 0;
	    #APP.PID_Kd := 0;
	    #APP.PID_ComponenteIntegrale := #JogVelocitaT*100;
	END_IF;
	//   
	// Arresto repentino
	// *****************
	IF (#APP.Tiro = 202) THEN
	    // Inizializzazione Fase 4
	    IF (#APP.ArrestoRepentinoOneShoot = 0) THEN
	        #APP.TimerArrestoRepentino := 0;
	        #APP.ArrestoRepentinoOneShoot := 1;
	    END_IF;
	    //
	    #APP.TimerArrestoRepentino := #APP.TimerArrestoRepentino + 1;
	    #APP.TiroMinimoArrestoRepentino := #TiroMinimoFase4T * 175/100;
	    //
	    IF (#APP.TiroPrecedente <= 100) THEN
	        #APP.TiroAppoggio := #APP.TiroPrecedente;
	    END_IF;
	    //
	    IF (#APP.TiroPrecedente > 100 & #APP.TiroPrecedente <= 200) THEN
	        #APP.TiroAppoggio := #APP.TiroPrecedente - 100;
	    END_IF;
	    //
	    IF (#APP.TiroAppoggio < #APP.TiroMinimoArrestoRepentino) THEN
	        #APP.TiroAppoggio := #APP.TiroMinimoArrestoRepentino;
	    END_IF;
	    //
	    #APP.SetpointTiro := ((#IngressoAnalogicoMaxT - #IngressoAnalogicoMinT) * #APP.TiroAppoggio / 100) + #IngressoAnalogicoMinT;
	    //   
	    #APP.PID_Kp := #PID_KpT;
	    #APP.PID_Ki := #PID_KiTransitoriT * 175/100;
	    #APP.PID_Kd := #PID_KdT;
	    //
	    #APP.TiroRichiesto := #APP.TiroAppoggio;
	END_IF;
	//
	// Regolatore PID standard 
	#APP.ErroreAttuale := (#BallerinoT-#APP.SetpointTiro);
	//
	// Componente proporzionale del regolatore          
	#APP.PID_ComponenteProporzionale := #APP.PID_Kp*#APP.ErroreAttuale;
	//
	// Componente integrale del regolatore
	#APP.PID_ComponenteIntegrale := #APP.PID_ComponenteIntegrale+#APP.PID_Ki*#APP.ErroreAttuale/10;
	//
	IF (#APP.PID_ComponenteIntegrale > #PID_LimiteSuperioreIntegrale AND #APP.Tiro <> 210) THEN
	    #APP.PID_ComponenteIntegrale := #PID_LimiteSuperioreIntegrale;
	END_IF;
	//
	IF (#APP.PID_ComponenteIntegrale > 25500 AND #APP.Tiro = 210) THEN
	    #APP.PID_ComponenteIntegrale := 25500;
	END_IF;
	//
	IF (#APP.PID_ComponenteIntegrale < #PID_LimiteInferioreIntegrale) THEN
	    #APP.PID_ComponenteIntegrale := #PID_LimiteInferioreIntegrale;
	END_IF;
	//
	// Componente derivativa del regolatore
	// PID_ComponenteDerivativa = 10*PID_Kd*(ErroreAttuale-ErrorePrecedente);
	
	#APP.PID_ComponenteDerivativa := 10*#APP.PID_Kd*(#BallerinoT-#APP.BallerinoPrecedente[2]);
	
	//#PID_ComponenteDerivativa := 10 * #PID_Kd * (#BallerinoT - #APP.BallPrec_2);
	//
	IF (#APP.PID_ComponenteDerivativa > #PID_LimiteSuperioreDerivativa) THEN
	    #APP.PID_ComponenteDerivativa := #PID_LimiteSuperioreDerivativa;
	END_IF;
	//
	IF (#APP.PID_ComponenteDerivativa < #PID_LimiteInferioreDerivativa) THEN
	    #APP.PID_ComponenteDerivativa := #PID_LimiteInferioreDerivativa;
	END_IF;
	//
	#APP.PID_Uscita := (#APP.PID_ComponenteProporzionale+#APP.PID_ComponenteIntegrale+#APP.PID_ComponenteDerivativa)/100 ; //Le costanti Kp, Ki e Kd sono espresse nel display in centesimi
	//
	IF (#APP.PID_Uscita > #PID_LimiteSuperioreUscita) THEN
	    #APP.PID_Uscita := #PID_LimiteSuperioreUscita;
	END_IF;
	//
	IF (#APP.PID_Uscita < #PID_LimiteInferioreUscita) THEN
	    #APP.PID_Uscita := #PID_LimiteInferioreUscita;
	END_IF;
	//
	IF (#APP.Tiro = 0) THEN
	    #APP.PID_Uscita := 0;
	END_IF;
	//
	// Aggiornamento valori precedenti  
	#APP.ErrorePrecedente := #APP.ErroreAttuale;
	//
	IF (#APP.Tiro <= 200) THEN
	    #APP.TiroPrecedente := #APP.Tiro;
	END_IF;
	//
	#APP.BallerinoPrecedente[2] := #APP.BallerinoPrecedente[1];
	#APP.BallerinoPrecedente[1] := #APP.BallerinoPrecedente[0];
	#APP.BallerinoPrecedente[0] := #BallerinoT;
	// #APP.BallPrec_2 := #APP.BallPrec_1;
	// #APP.BallPrec_1 := #APP.BallPrec_0;
	// #APP.BallPrec_0 := #BallerinoT;
	//
	// Attuazione delle uscite analogiche che vanno agli inverter
	#ValoreUscitaRulloVeloce := #APP.PID_Uscita;
	
	// Prestiro per PGSM e PGSA
	IF (#FunzionamentoM20T = 0) THEN
	    //
	    #APP.PrestiroRichiesto := INT_TO_DINT(#PrestiroT) * 500/255 + 100;
	    // Arrotonda sempre all'intero inferiore, a prescindere. Sommando 0.5 arrotondo all'intero piu vicino
	    #APP.PrestiroAppoggio := 0.5 + DINT_TO_REAL(#ValoreUscitaRulloVeloce * (#PrestiroMeccanicoNativoT + 100) / #APP.PrestiroRichiesto);
	    #APP.PrestiroAppoggio := #APP.PrestiroAppoggio + (#OffsetRulloLentoT - 10);
	    IF (#APP.PrestiroAppoggio > 255) THEN
	        #APP.PrestiroAppoggio := 255;
	    END_IF;
	    #ValoreUscitaRulloLento := REAL_TO_DINT(#APP.PrestiroAppoggio);
	END_IF;
	//
	// Tiro ballerino SCSP valvola proporzionale        
	IF (#FunzionamentoM20T = 1) THEN
	    #ValoreUscitaRulloLento := #PrestiroT;
	    IF (#ValoreUscitaRulloLento > 255) THEN
	        #ValoreUscitaRulloLento := 255;
	    END_IF;
	END_IF;
	                
	                
	
END_FUNCTION

FUNCTION "FC43_PreCarriageTechnoplat" : Void   // FC43, LAD
TITLE = HS40 standard prestretch management
{ S7_Optimized_Access := 'FALSE' }
AUTHOR : Robopac
VERSION : 0.0
// stored: AutoNumber false, IsIECCheckEnabled false, SetENOAutomatically false, UDAEnableTagReadback false
BEGIN

REGION Network 1: Timer for prestretch restart
